// TIA Portal V18 program export: 0 tag tables, 0 data types, 87 data blocks, 42 code blocks (in call order from the OBs), 0 instance data blocks

DATA_BLOCK "DiagnosticDataBlock"
{ S7_Optimized_Access := 'FALSE' }
VERSION : 0.1
   STRUCT 
      DP : Struct
         DPReadStatus : Int;
         Status : Array[0..1023] of Bool;
      END_STRUCT;
      Profinet : Struct
         PNReadStatus : Int;
         Status : Array[0..1023] of Bool;
      END_STRUCT;
   END_STRUCT;


BEGIN

END_DATA_BLOCK

DATA_BLOCK "Sys"
{ S7_Optimized_Access := 'FALSE' }
VERSION : 0.1
   STRUCT 
      COM : Struct
         AlwaysOFF : Bool;
         AlwaysON : Bool;
         FlashTime100mS : Bool;
         FlashTime200mS : Bool;
         FlashTime500mS : Bool;
         FlashTime1S : Bool;
         FlashTime2S : Bool;
         SpareBit : Bool;
         PLCRestarted : Bool;
      END_STRUCT;
      SpareB1 : Array[0..7] of Byte;
      DateTime : Struct
         Set : Date_And_Time;
         Read : Date_And_Time;
         Trigger : Bool;
         ReturnValueRead : Int;
         ReturnValueSet : Int;
      END_STRUCT;
      SpareB2 : Array[0..17] of Byte;
      ScanTime : Struct
         CyclePrevious : Int;
         CycleMax : Int;
         CycleMin : Int;
      END_STRUCT;
      RETVALI : Int;
      RETVALW : Word;
      VersionManagement : Struct
         ProductLineName : String;
         ProjectNumber : String[20];
         "PLC IP Addr" : Array[0..3] of UInt;
         "HMI IP Addr" : Array[0..3] of UInt;
         PLCVersion : Array[0..1] of UInt;
         HMIVersion : Array[0..1] of UInt;
         "TIA Version" : String;
         StationID : Int;
         HMIPageID : Int;
      END_STRUCT;
   END_STRUCT;


BEGIN
   COM.AlwaysOFF := FALSE;
   COM.AlwaysON := TRUE;
   COM.FlashTime100mS := TRUE;
   COM.FlashTime200mS := TRUE;
   COM.FlashTime500mS := FALSE;
   COM.FlashTime1S := FALSE;
   COM.FlashTime2S := TRUE;
   COM.SpareBit := FALSE;
   COM.PLCRestarted := TRUE;
   SpareB1[0] := 16#00;
   SpareB1[1] := 16#00;
   SpareB1[2] := 16#00;
   SpareB1[3] := 16#00;
   SpareB1[4] := 16#00;
   SpareB1[5] := 16#00;
   SpareB1[6] := 16#00;
   SpareB1[7] := 16#00;
   DateTime.Set := DT#1990-01-01-00:00:00;
   DateTime.Read := DT#2025-03-12-08:03:05.785;
   DateTime.Trigger := FALSE;
   DateTime.ReturnValueRead := 0;
   DateTime.ReturnValueSet := 0;
   SpareB2[0] := 16#00;
   SpareB2[1] := 16#00;
   SpareB2[2] := 16#00;
   SpareB2[3] := 16#00;
   SpareB2[4] := 16#00;
   SpareB2[5] := 16#00;
   SpareB2[6] := 16#00;
   SpareB2[7] := 16#00;
   SpareB2[8] := 16#00;
   SpareB2[9] := 16#00;
   SpareB2[10] := 16#00;
   SpareB2[11] := 16#00;
   SpareB2[12] := 16#00;
   SpareB2[13] := 16#00;
   SpareB2[14] := 16#00;
   SpareB2[15] := 16#00;
   SpareB2[16] := 16#00;
   SpareB2[17] := 16#00;
   ScanTime.CyclePrevious := 14;
   ScanTime.CycleMax := 23;
   ScanTime.CycleMin := 9;
   RETVALI := 0;
   RETVALW := 16#0000;
   VersionManagement.ProductLineName := 'Assembly Line';
   VersionManagement.ProjectNumber := 'SZ23055';
   VersionManagement."PLC IP Addr"[0] := 192;
   VersionManagement."PLC IP Addr"[1] := 168;
   VersionManagement."PLC IP Addr"[2] := 10;
   VersionManagement."PLC IP Addr"[3] := 10;
   VersionManagement."HMI IP Addr"[0] := 192;
   VersionManagement."HMI IP Addr"[1] := 168;
   VersionManagement."HMI IP Addr"[2] := 45;
   VersionManagement."HMI IP Addr"[3] := 11;
   VersionManagement.PLCVersion[0] := 1;
   VersionManagement.PLCVersion[1] := 0;
   VersionManagement.HMIVersion[0] := 1;
   VersionManagement.HMIVersion[1] := 0;
   VersionManagement."TIA Version" := 'TIA V18';
   VersionManagement.StationID := 10;
   VersionManagement.HMIPageID := 0;

END_DATA_BLOCK

DATA_BLOCK "ST10_FB_Tower_4Lamp_DB"
{ S7_Optimized_Access := 'TRUE' }
VERSION : 0.1
NON_RETAIN
"FB_Tower_4Lamp"

BEGIN

END_DATA_BLOCK

DATA_BLOCK "ST10_SysOutput"
{ S7_Optimized_Access := 'TRUE' }
VERSION : 0.1
NON_RETAIN
   VAR 
      oTowerLight : Struct
         Red : Bool;
         Yellow : Bool;
         Green : Bool;
         Blue : Bool;
      END_STRUCT;
      HMIButtonLight : Struct
         ControlOn : Bool;
         ControlOff : Bool;
         MachineStart : Bool;
         MachineStop : Bool;
         ResetButton : Bool;
         "Manual/Auto" : Bool;
         SafetyGateUnlock : Bool;
      END_STRUCT;
      BoxLight : Struct
         oMachineStartLight : Bool;
         oMachineStopLight : Bool;
         oResetLight : Bool;
         oSafetyGateUnlockLight : Bool;
      END_STRUCT;
      SafetyDoorCoil : Array[1..20] of Bool;
      MaterialDoorCoil : Array[1..20] of Bool;
   END_VAR


BEGIN
   HMIButtonLight.ControlOn := false;
   HMIButtonLight.MachineStart := false;
   HMIButtonLight.MachineStop := false;
   HMIButtonLight.ResetButton := false;
   HMIButtonLight."Manual/Auto" := false;
   HMIButtonLight.SafetyGateUnlock := false;

END_DATA_BLOCK

DATA_BLOCK "AutoProcessData"
{ S7_Optimized_Access := 'FALSE' }
VERSION : 0.1
   STRUCT 
      A_ScanRotate { S7_SetPoint := 'False'} : "ProcessData";
      F_Robot1Grip1 : "ProcessData";
      F_Robot1Grip2 : "ProcessData";
      B_Press1 : "ProcessData";
      C_Glue : "ProcessData";
      F_Robot2Grip1 : "ProcessData";
      F_Robot2Grip2 : "ProcessData";
      C_GlueNGBuffer : "ProcessData";
      C_MagnScanNGBuffer : "ProcessData";
      B_Press2 : "ProcessData";
      F_Robot3Grip1 : "ProcessData";
      F_Robot3Grip2 : "ProcessData";
      H_ShafeLine : "ProcessData";
      J_ShafeLine : "ProcessData";
      K_ShafeLine : "ProcessData";
      L_ShafeLine : "ProcessData";
      ClearData : "ProcessData";
      A_Table_1 : Array[1..10] of "TableProcessData";
      A_Table_2 : Array[1..10] of "TableProcessData";
      FixtureCode_A1 { S7_SetPoint := 'True'} : Array[1..10] of String[128];
      FixtureCode_A2 { S7_SetPoint := 'True'} : Array[1..10] of String[128];
      GlobalData : Struct
         Table1CodeOKFlag : Bool;
         Table2CodeOKFlag : Bool;
         Fixture1CodeOKFlag : Bool;
         Fixture2CodeOKFlag : Bool;
         Robot2GripperCodeOKFlag : Bool;
         Robot1GripperCodeOKFlag : Bool;
         Robot3GripperCodeOKFlag : Bool;
         Spare_8 : Bool;
         Spare_9 : Bool;
         Spare_10 : Bool;
         Spare_11 : Bool;
         Spare_12 : Bool;
         Spare_13 : Bool;
         Spare_14 : Bool;
         Spare_15 : Bool;
         Spare_16 : Bool;
         DataIndex { S7_SetPoint := 'True'} : Int;
         Robot1GripCodeStatus1 : Int;
         Robot1GripCodeStatus2 : Int;
         Robot1GripCodeStatus3 : Int;
         Robot1GripCodeStatus4 : Int;
         Robot2GripCodeStatus1 : Int;
         Robot2GripCodeStatus2 : Int;
         Robot2GripCodeStatus3 : Int;
         Robot2GripCodeStatus4 : Int;
         Robot3GripCodeStatus1 : Int;
         Robot3GripCodeStatus2 : Int;
         Robot3GripCodeStatus3 : Int;
         Robot3GripCodeStatus4 : Int;
         FixtureCode_A1Status1 : Int;
         FixtureCode_A1Status2 : Int;
         FixtureCode_A1Status3 : Int;
         FixtureCode_A1Status4 : Int;
         FixtureCode_A1Status5 : Int;
         FixtureCode_A1Status6 : Int;
         FixtureCode_A1Status7 : Int;
         FixtureCode_A1Status8 : Int;
         FixtureCode_A1Status9 : Int;
         FixtureCode_A1Status10 : Int;
         FixtureCode_A2Status1 : Int;
         FixtureCode_A2Status2 : Int;
         FixtureCode_A2Status3 : Int;
         FixtureCode_A2Status4 : Int;
         FixtureCode_A2Status5 : Int;
         FixtureCode_A2Status6 : Int;
         FixtureCode_A2Status7 : Int;
         FixtureCode_A2Status8 : Int;
         FixtureCode_A2Status9 : Int;
         FixtureCode_A2Status10 : Int;
         Spare : Array[1..332] of Byte;
      END_STRUCT;
      DataBuffer { S7_SetPoint := 'False'} : Array[1..30] of "ProcessData";
      GripperCode_R1 { S7_SetPoint := 'True'} : Array[1..10] of String[128];
      GripperCode_R2 { S7_SetPoint := 'True'} : Array[1..10] of String[128];
      GripperCode_R3 { S7_SetPoint := 'True'} : Array[1..10] of String[128];
   END_STRUCT;


BEGIN
   A_Table_1[1].Code := 'SZ23055-OP010-E-Compressor-ring1 Loading tooling-1';
   A_Table_1[2].Code := 'SZ23055-OP010-E-Compressor-ring1 Loading tooling-2';
   A_Table_2[1].Code := 'SZ23055-OP010-E-Compressor-ring2 Loading tooling-1$R';
   GlobalData.DataIndex := 1;

END_DATA_BLOCK

DATA_BLOCK "PalletRelease"
{ S7_Optimized_Access := 'FALSE' }
VERSION : 0.1
NON_RETAIN
   STRUCT 
      Buffer : Struct
         AskPallet : Bool;
         UnloadFlag : Bool;
      END_STRUCT;
      LaserMarking : Struct
         AskPallet : Bool;
         UnloadFlag : Bool;
      END_STRUCT;
      Print : Struct
         AskPallet : Bool;
         UnloadFlag : Bool;
      END_STRUCT;
      Spare : Struct
         AskPallet : Bool;
         UnloadFlag : Bool;
      END_STRUCT;
      Spare2 : Struct
         AskPallet : Bool;
         UnloadFlag : Bool;
      END_STRUCT;
      "Time" {InstructionName := 'TOF_TIME'; LibVersion := '1.0'; S7_SetPoint := 'False'} : Array[0..1] of TOF_TIME;
      LaserMarkingBuffer { S7_SetPoint := 'False'} : "LaserMarkingBuffer";
   END_STRUCT;


BEGIN

END_DATA_BLOCK

DATA_BLOCK "ST10_GlobalError"
{ S7_Optimized_Access := 'FALSE' }
VERSION : 0.1
   STRUCT 
      COM : Struct
         MainPneumaticPressure1NOK : Bool;
         MainPneumaticPressure2NOK : Bool;
         MainPneumaticPressure3NOK : Bool;
         StationNotInHP : Bool;
         CabinetTemperatureNotOk : Bool;
         CoolingUnitNotOk : Bool;
         RotateTablePositionNOK : Bool;
         RotateTableNotInPosition : Bool;
         StationHardwareError : Bool;
         ChangeStyleError : Bool;
         Reserve3 : Bool;
         Reserve4 : Bool;
         Reserve5 : Bool;
         Reserve6 : Bool;
         Reserve7 : Bool;
         Reserve8 : Bool;
         Reserve : Array[1..4, 0..15] of Bool;
      END_STRUCT;
      Hardware : Struct
         PNSlaveStation01 : Array[1..10] of Struct
            Error : Bool;
            Reserve1 : Bool;
            Reserve2 : Bool;
         END_STRUCT;
         COMM : Array[1..5] of Struct
            CommunicationError : Bool;
            NoReceive : Bool;
            ReceiveWrong : Bool;
            Reserve1 : Bool;
            Reserve2 : Bool;
         END_STRUCT;
         PNSlaveStation02 : Array[1..10] of Struct
            Error : Bool;
            Reserve1 : Bool;
            Reserve2 : Bool;
            Reserve3 : Bool;
         END_STRUCT;
         PNSlaveStation03 : Array[1..10] of Struct
            Error : Bool;
            Reserve1 : Bool;
            Reserve2 : Bool;
            Reserve3 : Bool;
         END_STRUCT;
         ValveIsland : Array[1..5] of Struct
            SystemError : Bool;
            OffLine : Bool;
            Reserve1 : Bool;
            Reserve2 : Bool;
         END_STRUCT;
      END_STRUCT;
      Safety : Struct
         "Robot 1 Estop" : Bool;
         "Robot 2 Estop" : Bool;
         HMIEstopPBActivated : Bool;
         TableEstopPB1Activated : Bool;
         TableEstopPB2Activated : Bool;
         TableEstopPB3Activated : Bool;
         TableEstopPB4Activated : Bool;
         TableEstopPB5Activated : Bool;
         TableEstopPB6Activated : Bool;
         EStopSafety : Bool;
         TableEstopPB7Activated : Bool;
         TableEstopPB8Activated : Bool;
         TableEstopPB9Activated : Bool;
         StoveEstopActivated : Bool;
         "Robot 3 Estop" : Bool;
         Reserve9 : Bool;
         Reserve : Array[1..4, 0..15] of Bool;
      END_STRUCT;
      SafetyDoor : Struct
         "Type" : Array[1..5] of Struct
            NotOk : Bool;
            OpenInRunning : Bool;
            Reserve1 : Bool;
            Reserve2 : Bool;
         END_STRUCT;
         No : Array[1..9] of Struct
            NotLock : Bool;
            Notlocked : Bool;
            NotClose : Bool;
            Reserve1 : Bool;
            Reserve2 : Bool;
         END_STRUCT;
         MaterialDoor : Struct
            NotLock_1 : Bool;
            NotClose_1 : Bool;
            NotLock_2 : Bool;
            NotClose_2 : Bool;
            NotLock_3 : Bool;
            NotClose_3 : Bool;
            NotLock_4 : Bool;
            NotClose_4 : Bool;
            NotLock_5 : Bool;
            NotClose_5 : Bool;
            NotLock_6 : Bool;
            NotClose_6 : Bool;
            NotLock_7 : Bool;
            NotClose_7 : Bool;
            NotLock_8 : Bool;
            NotClose_8 : Bool;
         END_STRUCT;
      END_STRUCT;
      LightCurtain : Array[1..5] of Struct
         ActivatedInRunning : Bool;
         ActivatedInRotTableRun : Bool;
         Error : Bool;
         Reserve1 : Bool;
         Reserve2 : Bool;
      END_STRUCT;
      Product : Array[1..5] of Struct
         TypeSelectionError : Bool;
         TypeWrong : Bool;
         NotforStation : Bool;
         TypeAutoChangeError : Bool;
         Reserve2 : Bool;
      END_STRUCT;
      Fixture : Array[1..10] of Struct
         PositionError : Bool;
         TypeError : Bool;
         Reserve1 : Bool;
         Reserve2 : Bool;
      END_STRUCT;
      Breaker : Struct
         Trip : Array[1..16] of Bool;
      END_STRUCT;
   END_STRUCT;


BEGIN

END_DATA_BLOCK

DATA_BLOCK "ST10_TipDB"
{ S7_Optimized_Access := 'FALSE' }
VERSION : 0.1
   STRUCT 
      Global : Struct
         "1" : Struct
            ControlOn : Bool;
            closesafetyDoor : Bool;
            LockSafetyDoor : Bool;
            SelectAutoMode : Bool;
            SelectManualMode : Bool;
            AutoModeRunning : Bool;
            SafetyDoorLocked : Bool;
            SaferyDoorNotLocked : Bool;
            GoWP : Bool;
            Reset : Bool;
         END_STRUCT;
         "2" : Array[0..15] of Bool;
         "3" : Array[0..15] of Bool;
         "4" : Array[0..15] of Bool;
         "5" : Struct
            FuncrionDeactive1 : Bool;
            FuncrionDeactive2 : Bool;
            FuncrionDeactive3 : Bool;
            FuncrionDeactive4 : Bool;
            FuncrionDeactive5 : Bool;
            FuncrionDeactive6 : Bool;
            FuncrionDeactive7 : Bool;
            FuncrionDeactive8 : Bool;
         END_STRUCT;
         "6" : Array[0..15] of Bool;
         "7" : Struct
            ScanMainPartDMC1 : Bool;
            ScanPartDMC2 : Bool;
            ScanPartDMC3 : Bool;
            ScanPartDMC4 : Bool;
            ScanPartDMC5 : Bool;
            ScanPartDMC6 : Bool;
            ScanPartDMC7 : Bool;
            ScanPartDMC8 : Bool;
         END_STRUCT;
         "8" : Array[0..15] of Bool;
         "9" : Array[0..15] of Bool;
         "10" : Array[0..15] of Bool;
      END_STRUCT;
      OP1 : Struct
         "Take off product" : Bool;
         "Put product" : Bool;
         "Please scan the code" : Bool;
         "Please apply Oil" : Bool;
         "Please take the O-ring" : Bool;
         "Please put in the powertrain" : Bool;
         Static_2 : Bool;
         "Please pre-screw" : Bool;
         Static_1 : Bool;
         Static_3 : Bool;
         "Please press the button_1" : Bool;
         Reset : Bool;
      END_STRUCT;
      OP2 : Struct
         Static_4 : Bool;
         Static_2 : Bool;
         Static_3 : Bool;
         "Please press the button" : Bool;
         "Please press the trigger" : Bool;
         "Please take the paint pen" : Bool;
         "Please put back the paint pen" : Bool;
         Static_1 : Bool;
         "Please remove the product" : Bool;
         "Please press the screw gun trigger" : Bool;
      END_STRUCT;
   END_STRUCT;


BEGIN

END_DATA_BLOCK

DATA_BLOCK "Parameter"
{ S7_Optimized_Access := 'TRUE' }
VERSION : 0.1
NON_RETAIN
   VAR RETAIN
      AxisRun : Struct
         Axis { S7_SetPoint := 'False'} : Array[1..15] of "ServoType_UDT";
      END_STRUCT;
      AxisNuw : Struct
         Axis { S7_SetPoint := 'False'} : Array[1..15] of "ServoType_UDT";
      END_STRUCT;
      AxisDisplay : Struct
         Axis { S7_SetPoint := 'False'} : Array[1..15] of "ServoType_UDT";
      END_STRUCT;
      AxisSave : Struct
         Axis { S7_SetPoint := 'False'} : Array[1..15] of "ServoType_UDT";
      END_STRUCT;
      AxisStore : Array[1..15] of Struct
         Axis { S7_SetPoint := 'False'} : Array[1..15] of "ServoType_UDT";
      END_STRUCT;
   END_VAR


BEGIN
   AxisRun.Axis[1].Pos1.Position := 3.419;
   AxisRun.Axis[1].Pos1.Speed := 10000;
   AxisRun.Axis[1].Pos1.Reached := FALSE;
   AxisRun.Axis[1].Pos2.Position := 48.386;
   AxisRun.Axis[1].Pos2.Speed := 10000;
   AxisRun.Axis[1].Pos2.Reached := FALSE;
   AxisRun.Axis[1].Pos3.Position := 93.294;
   AxisRun.Axis[1].Pos3.Speed := 10000;
   AxisRun.Axis[1].Pos3.Reached := FALSE;
   AxisRun.Axis[1].Pos4.Position := 138.335;
   AxisRun.Axis[1].Pos4.Speed := 10000;
   AxisRun.Axis[1].Pos4.Reached := FALSE;
   AxisRun.Axis[1].Pos5.Position := 183.464;
   AxisRun.Axis[1].Pos5.Speed := 10000;
   AxisRun.Axis[1].Pos5.Reached := FALSE;
   AxisRun.Axis[1].Pos6.Position := 228.443;
   AxisRun.Axis[1].Pos6.Speed := 10000;
   AxisRun.Axis[1].Pos6.Reached := FALSE;
   AxisRun.Axis[1].Pos7.Position := 273.535;
   AxisRun.Axis[1].Pos7.Speed := 10000;
   AxisRun.Axis[1].Pos7.Reached := FALSE;
   AxisRun.Axis[1].Pos8.Position := 318.25;
   AxisRun.Axis[1].Pos8.Speed := 10000;
   AxisRun.Axis[1].Pos8.Reached := FALSE;
   AxisRun.Axis[1].Pos9.Position := 0.0;
   AxisRun.Axis[1].Pos9.Speed := 0;
   AxisRun.Axis[1].Pos9.Reached := FALSE;
   AxisRun.Axis[1].Pos10.Position := 0.0;
   AxisRun.Axis[1].Pos10.Speed := 0;
   AxisRun.Axis[1].Pos10.Reached := FALSE;
   AxisRun.Axis[1].Pos11.Position := 0.0;
   AxisRun.Axis[1].Pos11.Speed := 0;
   AxisRun.Axis[1].Pos11.Reached := FALSE;
   AxisRun.Axis[1].Pos12.Position := 0.0;
   AxisRun.Axis[1].Pos12.Speed := 0;
   AxisRun.Axis[1].Pos12.Reached := FALSE;
   AxisRun.Axis[1].Pos13.Position := 0.0;
   AxisRun.Axis[1].Pos13.Speed := 0;
   AxisRun.Axis[1].Pos13.Reached := FALSE;
   AxisRun.Axis[1].Pos14.Position := 0.0;
   AxisRun.Axis[1].Pos14.Speed := 0;
   AxisRun.Axis[1].Pos14.Reached := FALSE;
   AxisRun.Axis[1].Pos15.Position := 0.0;
   AxisRun.Axis[1].Pos15.Speed := 0;
   AxisRun.Axis[1].Pos15.Reached := FALSE;
   AxisRun.Axis[1].Pos16.Position := 0.0;
   AxisRun.Axis[1].Pos16.Speed := 0;
   AxisRun.Axis[1].Pos16.Reached := FALSE;
   AxisRun.Axis[1].Pos17.Position := 0.0;
   AxisRun.Axis[1].Pos17.Speed := 0;
   AxisRun.Axis[1].Pos17.Reached := FALSE;
   AxisRun.Axis[1].Pos18.Position := 0.0;
   AxisRun.Axis[1].Pos18.Speed := 0;
   AxisRun.Axis[1].Pos18.Reached := FALSE;
   AxisRun.Axis[1].Pos19.Position := 0.0;
   AxisRun.Axis[1].Pos19.Speed := 0;
   AxisRun.Axis[1].Pos19.Reached := FALSE;
   AxisRun.Axis[1].Pos20.Position := 0.0;
   AxisRun.Axis[1].Pos20.Speed := 0;
   AxisRun.Axis[1].Pos20.Reached := FALSE;
   AxisRun.Axis[1].Pos21.Position := 0.0;
   AxisRun.Axis[1].Pos21.Speed := 0;
   AxisRun.Axis[1].Pos21.Reached := FALSE;
   AxisRun.Axis[1].Pos22.Position := 0.0;
   AxisRun.Axis[1].Pos22.Speed := 0;
   AxisRun.Axis[1].Pos22.Reached := FALSE;
   AxisRun.Axis[1].Pos23.Position := 0.0;
   AxisRun.Axis[1].Pos23.Speed := 0;
   AxisRun.Axis[1].Pos23.Reached := FALSE;
   AxisRun.Axis[1].Pos24.Position := 0.0;
   AxisRun.Axis[1].Pos24.Speed := 0;
   AxisRun.Axis[1].Pos24.Reached := FALSE;
   AxisRun.Axis[1].Pos25.Position := 0.0;
   AxisRun.Axis[1].Pos25.Speed := 0;
   AxisRun.Axis[1].Pos25.Reached := FALSE;
   AxisRun.Axis[1].Pos26.Position := 0.0;
   AxisRun.Axis[1].Pos26.Speed := 0;
   AxisRun.Axis[1].Pos26.Reached := FALSE;
   AxisRun.Axis[1].Pos27.Position := 0.0;
   AxisRun.Axis[1].Pos27.Speed := 0;
   AxisRun.Axis[1].Pos27.Reached := FALSE;
   AxisRun.Axis[1].Pos28.Position := 0.0;
   AxisRun.Axis[1].Pos28.Speed := 0;
   AxisRun.Axis[1].Pos28.Reached := FALSE;
   AxisRun.Axis[1].Pos29.Position := 0.0;
   AxisRun.Axis[1].Pos29.Speed := 0;
   AxisRun.Axis[1].Pos29.Reached := FALSE;
   AxisRun.Axis[1].Pos30.Position := 0.0;
   AxisRun.Axis[1].Pos30.Speed := 0;
   AxisRun.Axis[1].Pos30.Reached := FALSE;
   AxisRun.Axis[2].Pos1.Position := 0.0;
   AxisRun.Axis[2].Pos1.Speed := 10000;
   AxisRun.Axis[2].Pos1.Reached := FALSE;
   AxisRun.Axis[2].Pos2.Position := 450.0;
   AxisRun.Axis[2].Pos2.Speed := 10000;
   AxisRun.Axis[2].Pos2.Reached := FALSE;
   AxisRun.Axis[2].Pos3.Position := 900.0;
   AxisRun.Axis[2].Pos3.Speed := 10000;
   AxisRun.Axis[2].Pos3.Reached := FALSE;
   AxisRun.Axis[2].Pos4.Position := 135.0;
   AxisRun.Axis[2].Pos4.Speed := 10000;
   AxisRun.Axis[2].Pos4.Reached := FALSE;
   AxisRun.Axis[2].Pos5.Position := 180.0;
   AxisRun.Axis[2].Pos5.Speed := 10000;
   AxisRun.Axis[2].Pos5.Reached := FALSE;
   AxisRun.Axis[2].Pos6.Position := 225.0;
   AxisRun.Axis[2].Pos6.Speed := 10000;
   AxisRun.Axis[2].Pos6.Reached := FALSE;
   AxisRun.Axis[2].Pos7.Position := 270.0;
   AxisRun.Axis[2].Pos7.Speed := 10000;
   AxisRun.Axis[2].Pos7.Reached := FALSE;
   AxisRun.Axis[2].Pos8.Position := 315.0;
   AxisRun.Axis[2].Pos8.Speed := 10000;
   AxisRun.Axis[2].Pos8.Reached := FALSE;
   AxisRun.Axis[2].Pos9.Position := 0.0;
   AxisRun.Axis[2].Pos9.Speed := 0;
   AxisRun.Axis[2].Pos9.Reached := FALSE;
   AxisRun.Axis[2].Pos10.Position := 0.0;
   AxisRun.Axis[2].Pos10.Speed := 0;
   AxisRun.Axis[2].Pos10.Reached := FALSE;
   AxisRun.Axis[2].Pos11.Position := 0.0;
   AxisRun.Axis[2].Pos11.Speed := 0;
   AxisRun.Axis[2].Pos11.Reached := FALSE;
   AxisRun.Axis[2].Pos12.Position := 0.0;
   AxisRun.Axis[2].Pos12.Speed := 0;
   AxisRun.Axis[2].Pos12.Reached := FALSE;
   AxisRun.Axis[2].Pos13.Position := 0.0;
   AxisRun.Axis[2].Pos13.Speed := 0;
   AxisRun.Axis[2].Pos13.Reached := FALSE;
   AxisRun.Axis[2].Pos14.Position := 0.0;
   AxisRun.Axis[2].Pos14.Speed := 0;
   AxisRun.Axis[2].Pos14.Reached := FALSE;
   AxisRun.Axis[2].Pos15.Position := 0.0;
   AxisRun.Axis[2].Pos15.Speed := 0;
   AxisRun.Axis[2].Pos15.Reached := FALSE;
   AxisRun.Axis[2].Pos16.Position := 0.0;
   AxisRun.Axis[2].Pos16.Speed := 0;
   AxisRun.Axis[2].Pos16.Reached := FALSE;
   AxisRun.Axis[2].Pos17.Position := 0.0;
   AxisRun.Axis[2].Pos17.Speed := 0;
   AxisRun.Axis[2].Pos17.Reached := FALSE;
   AxisRun.Axis[2].Pos18.Position := 0.0;
   AxisRun.Axis[2].Pos18.Speed := 0;
   AxisRun.Axis[2].Pos18.Reached := FALSE;
   AxisRun.Axis[2].Pos19.Position := 0.0;
   AxisRun.Axis[2].Pos19.Speed := 0;
   AxisRun.Axis[2].Pos19.Reached := FALSE;
   AxisRun.Axis[2].Pos20.Position := 0.0;
   AxisRun.Axis[2].Pos20.Speed := 0;
   AxisRun.Axis[2].Pos20.Reached := FALSE;
   AxisRun.Axis[2].Pos21.Position := 0.0;
   AxisRun.Axis[2].Pos21.Speed := 0;
   AxisRun.Axis[2].Pos21.Reached := FALSE;
   AxisRun.Axis[2].Pos22.Position := 0.0;
   AxisRun.Axis[2].Pos22.Speed := 0;
   AxisRun.Axis[2].Pos22.Reached := FALSE;
   AxisRun.Axis[2].Pos23.Position := 0.0;
   AxisRun.Axis[2].Pos23.Speed := 0;
   AxisRun.Axis[2].Pos23.Reached := FALSE;
   AxisRun.Axis[2].Pos24.Position := 0.0;
   AxisRun.Axis[2].Pos24.Speed := 0;
   AxisRun.Axis[2].Pos24.Reached := FALSE;
   AxisRun.Axis[2].Pos25.Position := 0.0;
   AxisRun.Axis[2].Pos25.Speed := 0;
   AxisRun.Axis[2].Pos25.Reached := FALSE;
   AxisRun.Axis[2].Pos26.Position := 0.0;
   AxisRun.Axis[2].Pos26.Speed := 0;
   AxisRun.Axis[2].Pos26.Reached := FALSE;
   AxisRun.Axis[2].Pos27.Position := 0.0;
   AxisRun.Axis[2].Pos27.Speed := 0;
   AxisRun.Axis[2].Pos27.Reached := FALSE;
   AxisRun.Axis[2].Pos28.Position := 0.0;
   AxisRun.Axis[2].Pos28.Speed := 0;
   AxisRun.Axis[2].Pos28.Reached := FALSE;
   AxisRun.Axis[2].Pos29.Position := 0.0;
   AxisRun.Axis[2].Pos29.Speed := 0;
   AxisRun.Axis[2].Pos29.Reached := FALSE;
   AxisRun.Axis[2].Pos30.Position := 0.0;
   AxisRun.Axis[2].Pos30.Speed := 0;
   AxisRun.Axis[2].Pos30.Reached := FALSE;
   AxisRun.Axis[3].Pos1.Position := 0.0;
   AxisRun.Axis[3].Pos1.Speed := 20000;
   AxisRun.Axis[3].Pos1.Reached := FALSE;
   AxisRun.Axis[3].Pos2.Position := 490.0;
   AxisRun.Axis[3].Pos2.Speed := 10000;
   AxisRun.Axis[3].Pos2.Reached := FALSE;
   AxisRun.Axis[3].Pos3.Position := 490.0;
   AxisRun.Axis[3].Pos3.Speed := 10000;
   AxisRun.Axis[3].Pos3.Reached := FALSE;
   AxisRun.Axis[3].Pos4.Position := 490.0;
   AxisRun.Axis[3].Pos4.Speed := 10000;
   AxisRun.Axis[3].Pos4.Reached := FALSE;
   AxisRun.Axis[3].Pos5.Position := 0.0;
   AxisRun.Axis[3].Pos5.Speed := 0;
   AxisRun.Axis[3].Pos5.Reached := FALSE;
   AxisRun.Axis[3].Pos6.Position := 490.0;
   AxisRun.Axis[3].Pos6.Speed := 10000;
   AxisRun.Axis[3].Pos6.Reached := FALSE;
   AxisRun.Axis[3].Pos7.Position := 90.0;
   AxisRun.Axis[3].Pos7.Speed := 10000;
   AxisRun.Axis[3].Pos7.Reached := FALSE;
   AxisRun.Axis[3].Pos8.Position := 180.0;
   AxisRun.Axis[3].Pos8.Speed := 10000;
   AxisRun.Axis[3].Pos8.Reached := FALSE;
   AxisRun.Axis[3].Pos9.Position := 270.0;
   AxisRun.Axis[3].Pos9.Speed := 10000;
   AxisRun.Axis[3].Pos9.Reached := FALSE;
   AxisRun.Axis[3].Pos10.Position := 0.0;
   AxisRun.Axis[3].Pos10.Speed := 0;
   AxisRun.Axis[3].Pos10.Reached := FALSE;
   AxisRun.Axis[3].Pos11.Position := 0.0;
   AxisRun.Axis[3].Pos11.Speed := 0;
   AxisRun.Axis[3].Pos11.Reached := FALSE;
   AxisRun.Axis[3].Pos12.Position := 0.0;
   AxisRun.Axis[3].Pos12.Speed := 0;
   AxisRun.Axis[3].Pos12.Reached := FALSE;
   AxisRun.Axis[3].Pos13.Position := 0.0;
   AxisRun.Axis[3].Pos13.Speed := 0;
   AxisRun.Axis[3].Pos13.Reached := FALSE;
   AxisRun.Axis[3].Pos14.Position := 0.0;
   AxisRun.Axis[3].Pos14.Speed := 0;
   AxisRun.Axis[3].Pos14.Reached := FALSE;
   AxisRun.Axis[3].Pos15.Position := 0.0;
   AxisRun.Axis[3].Pos15.Speed := 0;
   AxisRun.Axis[3].Pos15.Reached := FALSE;
   AxisRun.Axis[3].Pos16.Position := 0.0;
   AxisRun.Axis[3].Pos16.Speed := 0;
   AxisRun.Axis[3].Pos16.Reached := FALSE;
   AxisRun.Axis[3].Pos17.Position := 0.0;
   AxisRun.Axis[3].Pos17.Speed := 0;
   AxisRun.Axis[3].Pos17.Reached := FALSE;
   AxisRun.Axis[3].Pos18.Position := 0.0;
   AxisRun.Axis[3].Pos18.Speed := 0;
   AxisRun.Axis[3].Pos18.Reached := FALSE;
   AxisRun.Axis[3].Pos19.Position := 0.0;
   AxisRun.Axis[3].Pos19.Speed := 0;
   AxisRun.Axis[3].Pos19.Reached := FALSE;
   AxisRun.Axis[3].Pos20.Position := 0.0;
   AxisRun.Axis[3].Pos20.Speed := 0;
   AxisRun.Axis[3].Pos20.Reached := FALSE;
   AxisRun.Axis[3].Pos21.Position := 0.0;
   AxisRun.Axis[3].Pos21.Speed := 0;
   AxisRun.Axis[3].Pos21.Reached := FALSE;
   AxisRun.Axis[3].Pos22.Position := 0.0;
   AxisRun.Axis[3].Pos22.Speed := 0;
   AxisRun.Axis[3].Pos22.Reached := FALSE;
   AxisRun.Axis[3].Pos23.Position := 0.0;
   AxisRun.Axis[3].Pos23.Speed := 0;
   AxisRun.Axis[3].Pos23.Reached := FALSE;
   AxisRun.Axis[3].Pos24.Position := 0.0;
   AxisRun.Axis[3].Pos24.Speed := 0;
   AxisRun.Axis[3].Pos24.Reached := FALSE;
   AxisRun.Axis[3].Pos25.Position := 0.0;
   AxisRun.Axis[3].Pos25.Speed := 0;
   AxisRun.Axis[3].Pos25.Reached := FALSE;
   AxisRun.Axis[3].Pos26.Position := 0.0;
   AxisRun.Axis[3].Pos26.Speed := 0;
   AxisRun.Axis[3].Pos26.Reached := FALSE;
   AxisRun.Axis[3].Pos27.Position := 0.0;
   AxisRun.Axis[3].Pos27.Speed := 0;
   AxisRun.Axis[3].Pos27.Reached := FALSE;
   AxisRun.Axis[3].Pos28.Position := 0.0;
   AxisRun.Axis[3].Pos28.Speed := 0;
   AxisRun.Axis[3].Pos28.Reached := FALSE;
   AxisRun.Axis[3].Pos29.Position := 0.0;
   AxisRun.Axis[3].Pos29.Speed := 0;
   AxisRun.Axis[3].Pos29.Reached := FALSE;
   AxisRun.Axis[3].Pos30.Position := 0.0;
   AxisRun.Axis[3].Pos30.Speed := 0;
   AxisRun.Axis[3].Pos30.Reached := FALSE;
   AxisRun.Axis[4].Pos1.Position := 3.585;
   AxisRun.Axis[4].Pos1.Speed := 10000;
   AxisRun.Axis[4].Pos1.Reached := FALSE;
   AxisRun.Axis[4].Pos2.Position := 48.61;
   AxisRun.Axis[4].Pos2.Speed := 10000;
   AxisRun.Axis[4].Pos2.Reached := FALSE;
   AxisRun.Axis[4].Pos3.Position := 93.637;
   AxisRun.Axis[4].Pos3.Speed := 10000;
   AxisRun.Axis[4].Pos3.Reached := FALSE;
   AxisRun.Axis[4].Pos4.Position := 138.606;
   AxisRun.Axis[4].Pos4.Speed := 10000;
   AxisRun.Axis[4].Pos4.Reached := FALSE;
   AxisRun.Axis[4].Pos5.Position := 183.388;
   AxisRun.Axis[4].Pos5.Speed := 10000;
   AxisRun.Axis[4].Pos5.Reached := FALSE;
   AxisRun.Axis[4].Pos6.Position := 228.458;
   AxisRun.Axis[4].Pos6.Speed := 10000;
   AxisRun.Axis[4].Pos6.Reached := FALSE;
   AxisRun.Axis[4].Pos7.Position := 273.513;
   AxisRun.Axis[4].Pos7.Speed := 10000;
   AxisRun.Axis[4].Pos7.Reached := FALSE;
   AxisRun.Axis[4].Pos8.Position := 318.501;
   AxisRun.Axis[4].Pos8.Speed := 10000;
   AxisRun.Axis[4].Pos8.Reached := FALSE;
   AxisRun.Axis[4].Pos9.Position := 0.0;
   AxisRun.Axis[4].Pos9.Speed := 0;
   AxisRun.Axis[4].Pos9.Reached := FALSE;
   AxisRun.Axis[4].Pos10.Position := 0.0;
   AxisRun.Axis[4].Pos10.Speed := 0;
   AxisRun.Axis[4].Pos10.Reached := FALSE;
   AxisRun.Axis[4].Pos11.Position := 0.0;
   AxisRun.Axis[4].Pos11.Speed := 0;
   AxisRun.Axis[4].Pos11.Reached := FALSE;
   AxisRun.Axis[4].Pos12.Position := 0.0;
   AxisRun.Axis[4].Pos12.Speed := 0;
   AxisRun.Axis[4].Pos12.Reached := FALSE;
   AxisRun.Axis[4].Pos13.Position := 0.0;
   AxisRun.Axis[4].Pos13.Speed := 0;
   AxisRun.Axis[4].Pos13.Reached := FALSE;
   AxisRun.Axis[4].Pos14.Position := 0.0;
   AxisRun.Axis[4].Pos14.Speed := 0;
   AxisRun.Axis[4].Pos14.Reached := FALSE;
   AxisRun.Axis[4].Pos15.Position := 0.0;
   AxisRun.Axis[4].Pos15.Speed := 0;
   AxisRun.Axis[4].Pos15.Reached := FALSE;
   AxisRun.Axis[4].Pos16.Position := 0.0;
   AxisRun.Axis[4].Pos16.Speed := 0;
   AxisRun.Axis[4].Pos16.Reached := FALSE;
   AxisRun.Axis[4].Pos17.Position := 0.0;
   AxisRun.Axis[4].Pos17.Speed := 0;
   AxisRun.Axis[4].Pos17.Reached := FALSE;
   AxisRun.Axis[4].Pos18.Position := 0.0;
   AxisRun.Axis[4].Pos18.Speed := 0;
   AxisRun.Axis[4].Pos18.Reached := FALSE;
   AxisRun.Axis[4].Pos19.Position := 0.0;
   AxisRun.Axis[4].Pos19.Speed := 0;
   AxisRun.Axis[4].Pos19.Reached := FALSE;
   AxisRun.Axis[4].Pos20.Position := 0.0;
   AxisRun.Axis[4].Pos20.Speed := 0;
   AxisRun.Axis[4].Pos20.Reached := FALSE;
   AxisRun.Axis[4].Pos21.Position := 0.0;
   AxisRun.Axis[4].Pos21.Speed := 0;
   AxisRun.Axis[4].Pos21.Reached := FALSE;
   AxisRun.Axis[4].Pos22.Position := 0.0;
   AxisRun.Axis[4].Pos22.Speed := 0;
   AxisRun.Axis[4].Pos22.Reached := FALSE;
   AxisRun.Axis[4].Pos23.Position := 0.0;
   AxisRun.Axis[4].Pos23.Speed := 0;
   AxisRun.Axis[4].Pos23.Reached := FALSE;
   AxisRun.Axis[4].Pos24.Position := 0.0;
   AxisRun.Axis[4].Pos24.Speed := 0;
   AxisRun.Axis[4].Pos24.Reached := FALSE;
   AxisRun.Axis[4].Pos25.Position := 0.0;
   AxisRun.Axis[4].Pos25.Speed := 0;
   AxisRun.Axis[4].Pos25.Reached := FALSE;
   AxisRun.Axis[4].Pos26.Position := 0.0;
   AxisRun.Axis[4].Pos26.Speed := 0;
   AxisRun.Axis[4].Pos26.Reached := FALSE;
   AxisRun.Axis[4].Pos27.Position := 0.0;
   AxisRun.Axis[4].Pos27.Speed := 0;
   AxisRun.Axis[4].Pos27.Reached := FALSE;
   AxisRun.Axis[4].Pos28.Position := 0.0;
   AxisRun.Axis[4].Pos28.Speed := 0;
   AxisRun.Axis[4].Pos28.Reached := FALSE;
   AxisRun.Axis[4].Pos29.Position := 0.0;
   AxisRun.Axis[4].Pos29.Speed := 0;
   AxisRun.Axis[4].Pos29.Reached := FALSE;
   AxisRun.Axis[4].Pos30.Position := 0.0;
   AxisRun.Axis[4].Pos30.Speed := 0;
   AxisRun.Axis[4].Pos30.Reached := FALSE;
   AxisRun.Axis[5].Pos1.Position := 143.76;
   AxisRun.Axis[5].Pos1.Speed := 200;
   AxisRun.Axis[5].Pos1.Reached := FALSE;
   AxisRun.Axis[5].Pos2.Position := 143.76;
   AxisRun.Axis[5].Pos2.Speed := 200;
   AxisRun.Axis[5].Pos2.Reached := FALSE;
   AxisRun.Axis[5].Pos3.Position := 137.76;
   AxisRun.Axis[5].Pos3.Speed := 200;
   AxisRun.Axis[5].Pos3.Reached := FALSE;
   AxisRun.Axis[5].Pos4.Position := 130.36;
   AxisRun.Axis[5].Pos4.Speed := 200;
   AxisRun.Axis[5].Pos4.Reached := FALSE;
   AxisRun.Axis[5].Pos5.Position := 124.16;
   AxisRun.Axis[5].Pos5.Speed := 200;
   AxisRun.Axis[5].Pos5.Reached := FALSE;
   AxisRun.Axis[5].Pos6.Position := 125.65;
   AxisRun.Axis[5].Pos6.Speed := 200;
   AxisRun.Axis[5].Pos6.Reached := FALSE;
   AxisRun.Axis[5].Pos7.Position := 48.11;
   AxisRun.Axis[5].Pos7.Speed := 200;
   AxisRun.Axis[5].Pos7.Reached := FALSE;
   AxisRun.Axis[5].Pos8.Position := 0.0;
   AxisRun.Axis[5].Pos8.Speed := 200;
   AxisRun.Axis[5].Pos8.Reached := FALSE;
   AxisRun.Axis[5].Pos9.Position := 48.11;
   AxisRun.Axis[5].Pos9.Speed := 200;
   AxisRun.Axis[5].Pos9.Reached := FALSE;
   AxisRun.Axis[5].Pos10.Position := 0.0;
   AxisRun.Axis[5].Pos10.Speed := 0;
   AxisRun.Axis[5].Pos10.Reached := FALSE;
   AxisRun.Axis[5].Pos11.Position := 0.0;
   AxisRun.Axis[5].Pos11.Speed := 0;
   AxisRun.Axis[5].Pos11.Reached := FALSE;
   AxisRun.Axis[5].Pos12.Position := 0.0;
   AxisRun.Axis[5].Pos12.Speed := 0;
   AxisRun.Axis[5].Pos12.Reached := FALSE;
   AxisRun.Axis[5].Pos13.Position := 0.0;
   AxisRun.Axis[5].Pos13.Speed := 0;
   AxisRun.Axis[5].Pos13.Reached := FALSE;
   AxisRun.Axis[5].Pos14.Position := 0.0;
   AxisRun.Axis[5].Pos14.Speed := 0;
   AxisRun.Axis[5].Pos14.Reached := FALSE;
   AxisRun.Axis[5].Pos15.Position := 0.0;
   AxisRun.Axis[5].Pos15.Speed := 0;
   AxisRun.Axis[5].Pos15.Reached := FALSE;
   AxisRun.Axis[5].Pos16.Position := 0.0;
   AxisRun.Axis[5].Pos16.Speed := 0;
   AxisRun.Axis[5].Pos16.Reached := FALSE;
   AxisRun.Axis[5].Pos17.Position := 0.0;
   AxisRun.Axis[5].Pos17.Speed := 0;
   AxisRun.Axis[5].Pos17.Reached := FALSE;
   AxisRun.Axis[5].Pos18.Position := 0.0;
   AxisRun.Axis[5].Pos18.Speed := 0;
   AxisRun.Axis[5].Pos18.Reached := FALSE;
   AxisRun.Axis[5].Pos19.Position := 0.0;
   AxisRun.Axis[5].Pos19.Speed := 0;
   AxisRun.Axis[5].Pos19.Reached := FALSE;
   AxisRun.Axis[5].Pos20.Position := 0.0;
   AxisRun.Axis[5].Pos20.Speed := 0;
   AxisRun.Axis[5].Pos20.Reached := FALSE;
   AxisRun.Axis[5].Pos21.Position := 0.0;
   AxisRun.Axis[5].Pos21.Speed := 0;
   AxisRun.Axis[5].Pos21.Reached := FALSE;
   AxisRun.Axis[5].Pos22.Position := 0.0;
   AxisRun.Axis[5].Pos22.Speed := 0;
   AxisRun.Axis[5].Pos22.Reached := FALSE;
   AxisRun.Axis[5].Pos23.Position := 0.0;
   AxisRun.Axis[5].Pos23.Speed := 0;
   AxisRun.Axis[5].Pos23.Reached := FALSE;
   AxisRun.Axis[5].Pos24.Position := 0.0;
   AxisRun.Axis[5].Pos24.Speed := 0;
   AxisRun.Axis[5].Pos24.Reached := FALSE;
   AxisRun.Axis[5].Pos25.Position := 0.0;
   AxisRun.Axis[5].Pos25.Speed := 0;
   AxisRun.Axis[5].Pos25.Reached := FALSE;
   AxisRun.Axis[5].Pos26.Position := 0.0;
   AxisRun.Axis[5].Pos26.Speed := 0;
   AxisRun.Axis[5].Pos26.Reached := FALSE;
   AxisRun.Axis[5].Pos27.Position := 0.0;
   AxisRun.Axis[5].Pos27.Speed := 0;
   AxisRun.Axis[5].Pos27.Reached := FALSE;
   AxisRun.Axis[5].Pos28.Position := 0.0;
   AxisRun.Axis[5].Pos28.Speed := 0;
   AxisRun.Axis[5].Pos28.Reached := FALSE;
   AxisRun.Axis[5].Pos29.Position := 0.0;
   AxisRun.Axis[5].Pos29.Speed := 0;
   AxisRun.Axis[5].Pos29.Reached := FALSE;
   AxisRun.Axis[5].Pos30.Position := 0.0;
   AxisRun.Axis[5].Pos30.Speed := 0;
   AxisRun.Axis[5].Pos30.Reached := FALSE;
   AxisRun.Axis[6].Pos1.Position := 2.34;
   AxisRun.Axis[6].Pos1.Speed := 200;
   AxisRun.Axis[6].Pos1.Reached := FALSE;
   AxisRun.Axis[6].Pos2.Position := 76.0;
   AxisRun.Axis[6].Pos2.Speed := 200;
   AxisRun.Axis[6].Pos2.Reached := FALSE;
   AxisRun.Axis[6].Pos3.Position := 84.69;
   AxisRun.Axis[6].Pos3.Speed := 200;
   AxisRun.Axis[6].Pos3.Reached := FALSE;
   AxisRun.Axis[6].Pos4.Position := 84.69;
   AxisRun.Axis[6].Pos4.Speed := 200;
   AxisRun.Axis[6].Pos4.Reached := FALSE;
   AxisRun.Axis[6].Pos5.Position := 84.69;
   AxisRun.Axis[6].Pos5.Speed := 200;
   AxisRun.Axis[6].Pos5.Reached := FALSE;
   AxisRun.Axis[6].Pos6.Position := 84.69;
   AxisRun.Axis[6].Pos6.Speed := 200;
   AxisRun.Axis[6].Pos6.Reached := FALSE;
   AxisRun.Axis[6].Pos7.Position := 85.0;
   AxisRun.Axis[6].Pos7.Speed := 200;
   AxisRun.Axis[6].Pos7.Reached := FALSE;
   AxisRun.Axis[6].Pos8.Position := 88.53;
   AxisRun.Axis[6].Pos8.Speed := 200;
   AxisRun.Axis[6].Pos8.Reached := FALSE;
   AxisRun.Axis[6].Pos9.Position := 0.0;
   AxisRun.Axis[6].Pos9.Speed := 0;
   AxisRun.Axis[6].Pos9.Reached := FALSE;
   AxisRun.Axis[6].Pos10.Position := 0.0;
   AxisRun.Axis[6].Pos10.Speed := 0;
   AxisRun.Axis[6].Pos10.Reached := FALSE;
   AxisRun.Axis[6].Pos11.Position := 0.0;
   AxisRun.Axis[6].Pos11.Speed := 0;
   AxisRun.Axis[6].Pos11.Reached := FALSE;
   AxisRun.Axis[6].Pos12.Position := 0.0;
   AxisRun.Axis[6].Pos12.Speed := 0;
   AxisRun.Axis[6].Pos12.Reached := FALSE;
   AxisRun.Axis[6].Pos13.Position := 0.0;
   AxisRun.Axis[6].Pos13.Speed := 0;
   AxisRun.Axis[6].Pos13.Reached := FALSE;
   AxisRun.Axis[6].Pos14.Position := 0.0;
   AxisRun.Axis[6].Pos14.Speed := 0;
   AxisRun.Axis[6].Pos14.Reached := FALSE;
   AxisRun.Axis[6].Pos15.Position := 0.0;
   AxisRun.Axis[6].Pos15.Speed := 0;
   AxisRun.Axis[6].Pos15.Reached := FALSE;
   AxisRun.Axis[6].Pos16.Position := 0.0;
   AxisRun.Axis[6].Pos16.Speed := 0;
   AxisRun.Axis[6].Pos16.Reached := FALSE;
   AxisRun.Axis[6].Pos17.Position := 0.0;
   AxisRun.Axis[6].Pos17.Speed := 0;
   AxisRun.Axis[6].Pos17.Reached := FALSE;
   AxisRun.Axis[6].Pos18.Position := 0.0;
   AxisRun.Axis[6].Pos18.Speed := 0;
   AxisRun.Axis[6].Pos18.Reached := FALSE;
   AxisRun.Axis[6].Pos19.Position := 0.0;
   AxisRun.Axis[6].Pos19.Speed := 0;
   AxisRun.Axis[6].Pos19.Reached := FALSE;
   AxisRun.Axis[6].Pos20.Position := 0.0;
   AxisRun.Axis[6].Pos20.Speed := 0;
   AxisRun.Axis[6].Pos20.Reached := FALSE;
   AxisRun.Axis[6].Pos21.Position := 0.0;
   AxisRun.Axis[6].Pos21.Speed := 0;
   AxisRun.Axis[6].Pos21.Reached := FALSE;
   AxisRun.Axis[6].Pos22.Position := 0.0;
   AxisRun.Axis[6].Pos22.Speed := 0;
   AxisRun.Axis[6].Pos22.Reached := FALSE;
   AxisRun.Axis[6].Pos23.Position := 0.0;
   AxisRun.Axis[6].Pos23.Speed := 0;
   AxisRun.Axis[6].Pos23.Reached := FALSE;
   AxisRun.Axis[6].Pos24.Position := 0.0;
   AxisRun.Axis[6].Pos24.Speed := 0;
   AxisRun.Axis[6].Pos24.Reached := FALSE;
   AxisRun.Axis[6].Pos25.Position := 0.0;
   AxisRun.Axis[6].Pos25.Speed := 0;
   AxisRun.Axis[6].Pos25.Reached := FALSE;
   AxisRun.Axis[6].Pos26.Position := 0.0;
   AxisRun.Axis[6].Pos26.Speed := 0;
   AxisRun.Axis[6].Pos26.Reached := FALSE;
   AxisRun.Axis[6].Pos27.Position := 0.0;
   AxisRun.Axis[6].Pos27.Speed := 0;
   AxisRun.Axis[6].Pos27.Reached := FALSE;
   AxisRun.Axis[6].Pos28.Position := 0.0;
   AxisRun.Axis[6].Pos28.Speed := 0;
   AxisRun.Axis[6].Pos28.Reached := FALSE;
   AxisRun.Axis[6].Pos29.Position := 0.0;
   AxisRun.Axis[6].Pos29.Speed := 0;
   AxisRun.Axis[6].Pos29.Reached := FALSE;
   AxisRun.Axis[6].Pos30.Position := 0.0;
   AxisRun.Axis[6].Pos30.Speed := 0;
   AxisRun.Axis[6].Pos30.Reached := FALSE;
   AxisRun.Axis[7].Pos1.Position := 115.47;
   AxisRun.Axis[7].Pos1.Speed := 200;
   AxisRun.Axis[7].Pos1.Reached := FALSE;
   AxisRun.Axis[7].Pos2.Position := 115.47;
   AxisRun.Axis[7].Pos2.Speed := 200;
   AxisRun.Axis[7].Pos2.Reached := FALSE;
   AxisRun.Axis[7].Pos3.Position := 115.47;
   AxisRun.Axis[7].Pos3.Speed := 200;
   AxisRun.Axis[7].Pos3.Reached := FALSE;
   AxisRun.Axis[7].Pos4.Position := 115.47;
   AxisRun.Axis[7].Pos4.Speed := 200;
   AxisRun.Axis[7].Pos4.Reached := FALSE;
   AxisRun.Axis[7].Pos5.Position := 115.47;
   AxisRun.Axis[7].Pos5.Speed := 200;
   AxisRun.Axis[7].Pos5.Reached := FALSE;
   AxisRun.Axis[7].Pos6.Position := 110.18;
   AxisRun.Axis[7].Pos6.Speed := 200;
   AxisRun.Axis[7].Pos6.Reached := FALSE;
   AxisRun.Axis[7].Pos7.Position := 60.52;
   AxisRun.Axis[7].Pos7.Speed := 200;
   AxisRun.Axis[7].Pos7.Reached := FALSE;
   AxisRun.Axis[7].Pos8.Position := 80.0;
   AxisRun.Axis[7].Pos8.Speed := 100;
   AxisRun.Axis[7].Pos8.Reached := FALSE;
   AxisRun.Axis[7].Pos9.Position := 0.0;
   AxisRun.Axis[7].Pos9.Speed := 0;
   AxisRun.Axis[7].Pos9.Reached := FALSE;
   AxisRun.Axis[7].Pos10.Position := 0.0;
   AxisRun.Axis[7].Pos10.Speed := 0;
   AxisRun.Axis[7].Pos10.Reached := FALSE;
   AxisRun.Axis[7].Pos11.Position := 0.0;
   AxisRun.Axis[7].Pos11.Speed := 0;
   AxisRun.Axis[7].Pos11.Reached := FALSE;
   AxisRun.Axis[7].Pos12.Position := 0.0;
   AxisRun.Axis[7].Pos12.Speed := 0;
   AxisRun.Axis[7].Pos12.Reached := FALSE;
   AxisRun.Axis[7].Pos13.Position := 0.0;
   AxisRun.Axis[7].Pos13.Speed := 0;
   AxisRun.Axis[7].Pos13.Reached := FALSE;
   AxisRun.Axis[7].Pos14.Position := 0.0;
   AxisRun.Axis[7].Pos14.Speed := 0;
   AxisRun.Axis[7].Pos14.Reached := FALSE;
   AxisRun.Axis[7].Pos15.Position := 0.0;
   AxisRun.Axis[7].Pos15.Speed := 0;
   AxisRun.Axis[7].Pos15.Reached := FALSE;
   AxisRun.Axis[7].Pos16.Position := 0.0;
   AxisRun.Axis[7].Pos16.Speed := 0;
   AxisRun.Axis[7].Pos16.Reached := FALSE;
   AxisRun.Axis[7].Pos17.Position := 0.0;
   AxisRun.Axis[7].Pos17.Speed := 0;
   AxisRun.Axis[7].Pos17.Reached := FALSE;
   AxisRun.Axis[7].Pos18.Position := 0.0;
   AxisRun.Axis[7].Pos18.Speed := 0;
   AxisRun.Axis[7].Pos18.Reached := FALSE;
   AxisRun.Axis[7].Pos19.Position := 0.0;
   AxisRun.Axis[7].Pos19.Speed := 0;
   AxisRun.Axis[7].Pos19.Reached := FALSE;
   AxisRun.Axis[7].Pos20.Position := 0.0;
   AxisRun.Axis[7].Pos20.Speed := 0;
   AxisRun.Axis[7].Pos20.Reached := FALSE;
   AxisRun.Axis[7].Pos21.Position := 0.0;
   AxisRun.Axis[7].Pos21.Speed := 0;
   AxisRun.Axis[7].Pos21.Reached := FALSE;
   AxisRun.Axis[7].Pos22.Position := 0.0;
   AxisRun.Axis[7].Pos22.Speed := 0;
   AxisRun.Axis[7].Pos22.Reached := FALSE;
   AxisRun.Axis[7].Pos23.Position := 0.0;
   AxisRun.Axis[7].Pos23.Speed := 0;
   AxisRun.Axis[7].Pos23.Reached := FALSE;
   AxisRun.Axis[7].Pos24.Position := 0.0;
   AxisRun.Axis[7].Pos24.Speed := 0;
   AxisRun.Axis[7].Pos24.Reached := FALSE;
   AxisRun.Axis[7].Pos25.Position := 0.0;
   AxisRun.Axis[7].Pos25.Speed := 0;
   AxisRun.Axis[7].Pos25.Reached := FALSE;
   AxisRun.Axis[7].Pos26.Position := 0.0;
   AxisRun.Axis[7].Pos26.Speed := 0;
   AxisRun.Axis[7].Pos26.Reached := FALSE;
   AxisRun.Axis[7].Pos27.Position := 0.0;
   AxisRun.Axis[7].Pos27.Speed := 0;
   AxisRun.Axis[7].Pos27.Reached := FALSE;
   AxisRun.Axis[7].Pos28.Position := 0.0;
   AxisRun.Axis[7].Pos28.Speed := 0;
   AxisRun.Axis[7].Pos28.Reached := FALSE;
   AxisRun.Axis[7].Pos29.Position := 0.0;
   AxisRun.Axis[7].Pos29.Speed := 0;
   AxisRun.Axis[7].Pos29.Reached := FALSE;
   AxisRun.Axis[7].Pos30.Position := 0.0;
   AxisRun.Axis[7].Pos30.Speed := 0;
   AxisRun.Axis[7].Pos30.Reached := FALSE;
   AxisRun.Axis[8].Pos1.Position := 0.0;
   AxisRun.Axis[8].Pos1.Speed := 0;
   AxisRun.Axis[8].Pos1.Reached := FALSE;
   AxisRun.Axis[8].Pos2.Position := 0.0;
   AxisRun.Axis[8].Pos2.Speed := 0;
   AxisRun.Axis[8].Pos2.Reached := FALSE;
   AxisRun.Axis[8].Pos3.Position := 0.0;
   AxisRun.Axis[8].Pos3.Speed := 0;
   AxisRun.Axis[8].Pos3.Reached := FALSE;
   AxisRun.Axis[8].Pos4.Position := 0.0;
   AxisRun.Axis[8].Pos4.Speed := 0;
   AxisRun.Axis[8].Pos4.Reached := FALSE;
   AxisRun.Axis[8].Pos5.Position := 0.0;
   AxisRun.Axis[8].Pos5.Speed := 0;
   AxisRun.Axis[8].Pos5.Reached := FALSE;
   AxisRun.Axis[8].Pos6.Position := 0.0;
   AxisRun.Axis[8].Pos6.Speed := 0;
   AxisRun.Axis[8].Pos6.Reached := FALSE;
   AxisRun.Axis[8].Pos7.Position := 0.0;
   AxisRun.Axis[8].Pos7.Speed := 0;
   AxisRun.Axis[8].Pos7.Reached := FALSE;
   AxisRun.Axis[8].Pos8.Position := 0.0;
   AxisRun.Axis[8].Pos8.Speed := 0;
   AxisRun.Axis[8].Pos8.Reached := FALSE;
   AxisRun.Axis[8].Pos9.Position := 0.0;
   AxisRun.Axis[8].Pos9.Speed := 0;
   AxisRun.Axis[8].Pos9.Reached := FALSE;
   AxisRun.Axis[8].Pos10.Position := 0.0;
   AxisRun.Axis[8].Pos10.Speed := 0;
   AxisRun.Axis[8].Pos10.Reached := FALSE;
   AxisRun.Axis[8].Pos11.Position := 0.0;
   AxisRun.Axis[8].Pos11.Speed := 0;
   AxisRun.Axis[8].Pos11.Reached := FALSE;
   AxisRun.Axis[8].Pos12.Position := 0.0;
   AxisRun.Axis[8].Pos12.Speed := 0;
   AxisRun.Axis[8].Pos12.Reached := FALSE;
   AxisRun.Axis[8].Pos13.Position := 0.0;
   AxisRun.Axis[8].Pos13.Speed := 0;
   AxisRun.Axis[8].Pos13.Reached := FALSE;
   AxisRun.Axis[8].Pos14.Position := 0.0;
   AxisRun.Axis[8].Pos14.Speed := 0;
   AxisRun.Axis[8].Pos14.Reached := FALSE;
   AxisRun.Axis[8].Pos15.Position := 0.0;
   AxisRun.Axis[8].Pos15.Speed := 0;
   AxisRun.Axis[8].Pos15.Reached := FALSE;
   AxisRun.Axis[8].Pos16.Position := 0.0;
   AxisRun.Axis[8].Pos16.Speed := 0;
   AxisRun.Axis[8].Pos16.Reached := FALSE;
   AxisRun.Axis[8].Pos17.Position := 0.0;
   AxisRun.Axis[8].Pos17.Speed := 0;
   AxisRun.Axis[8].Pos17.Reached := FALSE;
   AxisRun.Axis[8].Pos18.Position := 0.0;
   AxisRun.Axis[8].Pos18.Speed := 0;
   AxisRun.Axis[8].Pos18.Reached := FALSE;
   AxisRun.Axis[8].Pos19.Position := 0.0;
   AxisRun.Axis[8].Pos19.Speed := 0;
   AxisRun.Axis[8].Pos19.Reached := FALSE;
   AxisRun.Axis[8].Pos20.Position := 0.0;
   AxisRun.Axis[8].Pos20.Speed := 0;
   AxisRun.Axis[8].Pos20.Reached := FALSE;
   AxisRun.Axis[8].Pos21.Position := 0.0;
   AxisRun.Axis[8].Pos21.Speed := 0;
   AxisRun.Axis[8].Pos21.Reached := FALSE;
   AxisRun.Axis[8].Pos22.Position := 0.0;
   AxisRun.Axis[8].Pos22.Speed := 0;
   AxisRun.Axis[8].Pos22.Reached := FALSE;
   AxisRun.Axis[8].Pos23.Position := 0.0;
   AxisRun.Axis[8].Pos23.Speed := 0;
   AxisRun.Axis[8].Pos23.Reached := FALSE;
   AxisRun.Axis[8].Pos24.Position := 0.0;
   AxisRun.Axis[8].Pos24.Speed := 0;
   AxisRun.Axis[8].Pos24.Reached := FALSE;
   AxisRun.Axis[8].Pos25.Position := 0.0;
   AxisRun.Axis[8].Pos25.Speed := 0;
   AxisRun.Axis[8].Pos25.Reached := FALSE;
   AxisRun.Axis[8].Pos26.Position := 0.0;
   AxisRun.Axis[8].Pos26.Speed := 0;
   AxisRun.Axis[8].Pos26.Reached := FALSE;
   AxisRun.Axis[8].Pos27.Position := 0.0;
   AxisRun.Axis[8].Pos27.Speed := 0;
   AxisRun.Axis[8].Pos27.Reached := FALSE;
   AxisRun.Axis[8].Pos28.Position := 0.0;
   AxisRun.Axis[8].Pos28.Speed := 0;
   AxisRun.Axis[8].Pos28.Reached := FALSE;
   AxisRun.Axis[8].Pos29.Position := 0.0;
   AxisRun.Axis[8].Pos29.Speed := 0;
   AxisRun.Axis[8].Pos29.Reached := FALSE;
   AxisRun.Axis[8].Pos30.Position := 0.0;
   AxisRun.Axis[8].Pos30.Speed := 0;
   AxisRun.Axis[8].Pos30.Reached := FALSE;
   AxisRun.Axis[9].Pos1.Position := 0.0;
   AxisRun.Axis[9].Pos1.Speed := 0;
   AxisRun.Axis[9].Pos1.Reached := FALSE;
   AxisRun.Axis[9].Pos2.Position := 0.0;
   AxisRun.Axis[9].Pos2.Speed := 0;
   AxisRun.Axis[9].Pos2.Reached := FALSE;
   AxisRun.Axis[9].Pos3.Position := 0.0;
   AxisRun.Axis[9].Pos3.Speed := 0;
   AxisRun.Axis[9].Pos3.Reached := FALSE;
   AxisRun.Axis[9].Pos4.Position := 0.0;
   AxisRun.Axis[9].Pos4.Speed := 0;
   AxisRun.Axis[9].Pos4.Reached := FALSE;
   AxisRun.Axis[9].Pos5.Position := 0.0;
   AxisRun.Axis[9].Pos5.Speed := 0;
   AxisRun.Axis[9].Pos5.Reached := FALSE;
   AxisRun.Axis[9].Pos6.Position := 0.0;
   AxisRun.Axis[9].Pos6.Speed := 0;
   AxisRun.Axis[9].Pos6.Reached := FALSE;
   AxisRun.Axis[9].Pos7.Position := 0.0;
   AxisRun.Axis[9].Pos7.Speed := 0;
   AxisRun.Axis[9].Pos7.Reached := FALSE;
   AxisRun.Axis[9].Pos8.Position := 0.0;
   AxisRun.Axis[9].Pos8.Speed := 0;
   AxisRun.Axis[9].Pos8.Reached := FALSE;
   AxisRun.Axis[9].Pos9.Position := 0.0;
   AxisRun.Axis[9].Pos9.Speed := 0;
   AxisRun.Axis[9].Pos9.Reached := FALSE;
   AxisRun.Axis[9].Pos10.Position := 0.0;
   AxisRun.Axis[9].Pos10.Speed := 0;
   AxisRun.Axis[9].Pos10.Reached := FALSE;
   AxisRun.Axis[9].Pos11.Position := 0.0;
   AxisRun.Axis[9].Pos11.Speed := 0;
   AxisRun.Axis[9].Pos11.Reached := FALSE;
   AxisRun.Axis[9].Pos12.Position := 0.0;
   AxisRun.Axis[9].Pos12.Speed := 0;
   AxisRun.Axis[9].Pos12.Reached := FALSE;
   AxisRun.Axis[9].Pos13.Position := 0.0;
   AxisRun.Axis[9].Pos13.Speed := 0;
   AxisRun.Axis[9].Pos13.Reached := FALSE;
   AxisRun.Axis[9].Pos14.Position := 0.0;
   AxisRun.Axis[9].Pos14.Speed := 0;
   AxisRun.Axis[9].Pos14.Reached := FALSE;
   AxisRun.Axis[9].Pos15.Position := 0.0;
   AxisRun.Axis[9].Pos15.Speed := 0;
   AxisRun.Axis[9].Pos15.Reached := FALSE;
   AxisRun.Axis[9].Pos16.Position := 0.0;
   AxisRun.Axis[9].Pos16.Speed := 0;
   AxisRun.Axis[9].Pos16.Reached := FALSE;
   AxisRun.Axis[9].Pos17.Position := 0.0;
   AxisRun.Axis[9].Pos17.Speed := 0;
   AxisRun.Axis[9].Pos17.Reached := FALSE;
   AxisRun.Axis[9].Pos18.Position := 0.0;
   AxisRun.Axis[9].Pos18.Speed := 0;
   AxisRun.Axis[9].Pos18.Reached := FALSE;
   AxisRun.Axis[9].Pos19.Position := 0.0;
   AxisRun.Axis[9].Pos19.Speed := 0;
   AxisRun.Axis[9].Pos19.Reached := FALSE;
   AxisRun.Axis[9].Pos20.Position := 0.0;
   AxisRun.Axis[9].Pos20.Speed := 0;
   AxisRun.Axis[9].Pos20.Reached := FALSE;
   AxisRun.Axis[9].Pos21.Position := 0.0;
   AxisRun.Axis[9].Pos21.Speed := 0;
   AxisRun.Axis[9].Pos21.Reached := FALSE;
   AxisRun.Axis[9].Pos22.Position := 0.0;
   AxisRun.Axis[9].Pos22.Speed := 0;
   AxisRun.Axis[9].Pos22.Reached := FALSE;
   AxisRun.Axis[9].Pos23.Position := 0.0;
   AxisRun.Axis[9].Pos23.Speed := 0;
   AxisRun.Axis[9].Pos23.Reached := FALSE;
   AxisRun.Axis[9].Pos24.Position := 0.0;
   AxisRun.Axis[9].Pos24.Speed := 0;
   AxisRun.Axis[9].Pos24.Reached := FALSE;
   AxisRun.Axis[9].Pos25.Position := 0.0;
   AxisRun.Axis[9].Pos25.Speed := 0;
   AxisRun.Axis[9].Pos25.Reached := FALSE;
   AxisRun.Axis[9].Pos26.Position := 0.0;
   AxisRun.Axis[9].Pos26.Speed := 0;
   AxisRun.Axis[9].Pos26.Reached := FALSE;
   AxisRun.Axis[9].Pos27.Position := 0.0;
   AxisRun.Axis[9].Pos27.Speed := 0;
   AxisRun.Axis[9].Pos27.Reached := FALSE;
   AxisRun.Axis[9].Pos28.Position := 0.0;
   AxisRun.Axis[9].Pos28.Speed := 0;
   AxisRun.Axis[9].Pos28.Reached := FALSE;
   AxisRun.Axis[9].Pos29.Position := 0.0;
   AxisRun.Axis[9].Pos29.Speed := 0;
   AxisRun.Axis[9].Pos29.Reached := FALSE;
   AxisRun.Axis[9].Pos30.Position := 0.0;
   AxisRun.Axis[9].Pos30.Speed := 0;
   AxisRun.Axis[9].Pos30.Reached := FALSE;
   AxisRun.Axis[10].Pos1.Position := 0.0;
   AxisRun.Axis[10].Pos1.Speed := 0;
   AxisRun.Axis[10].Pos1.Reached := FALSE;
   AxisRun.Axis[10].Pos2.Position := 0.0;
   AxisRun.Axis[10].Pos2.Speed := 0;
   AxisRun.Axis[10].Pos2.Reached := FALSE;
   AxisRun.Axis[10].Pos3.Position := 0.0;
   AxisRun.Axis[10].Pos3.Speed := 0;
   AxisRun.Axis[10].Pos3.Reached := FALSE;
   AxisRun.Axis[10].Pos4.Position := 0.0;
   AxisRun.Axis[10].Pos4.Speed := 0;
   AxisRun.Axis[10].Pos4.Reached := FALSE;
   AxisRun.Axis[10].Pos5.Position := 0.0;
   AxisRun.Axis[10].Pos5.Speed := 0;
   AxisRun.Axis[10].Pos5.Reached := FALSE;
   AxisRun.Axis[10].Pos6.Position := 0.0;
   AxisRun.Axis[10].Pos6.Speed := 0;
   AxisRun.Axis[10].Pos6.Reached := FALSE;
   AxisRun.Axis[10].Pos7.Position := 0.0;
   AxisRun.Axis[10].Pos7.Speed := 0;
   AxisRun.Axis[10].Pos7.Reached := FALSE;
   AxisRun.Axis[10].Pos8.Position := 0.0;
   AxisRun.Axis[10].Pos8.Speed := 0;
   AxisRun.Axis[10].Pos8.Reached := FALSE;
   AxisRun.Axis[10].Pos9.Position := 0.0;
   AxisRun.Axis[10].Pos9.Speed := 0;
   AxisRun.Axis[10].Pos9.Reached := FALSE;
   AxisRun.Axis[10].Pos10.Position := 0.0;
   AxisRun.Axis[10].Pos10.Speed := 0;
   AxisRun.Axis[10].Pos10.Reached := FALSE;
   AxisRun.Axis[10].Pos11.Position := 0.0;
   AxisRun.Axis[10].Pos11.Speed := 0;
   AxisRun.Axis[10].Pos11.Reached := FALSE;
   AxisRun.Axis[10].Pos12.Position := 0.0;
   AxisRun.Axis[10].Pos12.Speed := 0;
   AxisRun.Axis[10].Pos12.Reached := FALSE;
   AxisRun.Axis[10].Pos13.Position := 0.0;
   AxisRun.Axis[10].Pos13.Speed := 0;
   AxisRun.Axis[10].Pos13.Reached := FALSE;
   AxisRun.Axis[10].Pos14.Position := 0.0;
   AxisRun.Axis[10].Pos14.Speed := 0;
   AxisRun.Axis[10].Pos14.Reached := FALSE;
   AxisRun.Axis[10].Pos15.Position := 0.0;
   AxisRun.Axis[10].Pos15.Speed := 0;
   AxisRun.Axis[10].Pos15.Reached := FALSE;
   AxisRun.Axis[10].Pos16.Position := 0.0;
   AxisRun.Axis[10].Pos16.Speed := 0;
   AxisRun.Axis[10].Pos16.Reached := FALSE;
   AxisRun.Axis[10].Pos17.Position := 0.0;
   AxisRun.Axis[10].Pos17.Speed := 0;
   AxisRun.Axis[10].Pos17.Reached := FALSE;
   AxisRun.Axis[10].Pos18.Position := 0.0;
   AxisRun.Axis[10].Pos18.Speed := 0;
   AxisRun.Axis[10].Pos18.Reached := FALSE;
   AxisRun.Axis[10].Pos19.Position := 0.0;
   AxisRun.Axis[10].Pos19.Speed := 0;
   AxisRun.Axis[10].Pos19.Reached := FALSE;
   AxisRun.Axis[10].Pos20.Position := 0.0;
   AxisRun.Axis[10].Pos20.Speed := 0;
   AxisRun.Axis[10].Pos20.Reached := FALSE;
   AxisRun.Axis[10].Pos21.Position := 0.0;
   AxisRun.Axis[10].Pos21.Speed := 0;
   AxisRun.Axis[10].Pos21.Reached := FALSE;
   AxisRun.Axis[10].Pos22.Position := 0.0;
   AxisRun.Axis[10].Pos22.Speed := 0;
   AxisRun.Axis[10].Pos22.Reached := FALSE;
   AxisRun.Axis[10].Pos23.Position := 0.0;
   AxisRun.Axis[10].Pos23.Speed := 0;
   AxisRun.Axis[10].Pos23.Reached := FALSE;
   AxisRun.Axis[10].Pos24.Position := 0.0;
   AxisRun.Axis[10].Pos24.Speed := 0;
   AxisRun.Axis[10].Pos24.Reached := FALSE;
   AxisRun.Axis[10].Pos25.Position := 0.0;
   AxisRun.Axis[10].Pos25.Speed := 0;
   AxisRun.Axis[10].Pos25.Reached := FALSE;
   AxisRun.Axis[10].Pos26.Position := 0.0;
   AxisRun.Axis[10].Pos26.Speed := 0;
   AxisRun.Axis[10].Pos26.Reached := FALSE;
   AxisRun.Axis[10].Pos27.Position := 0.0;
   AxisRun.Axis[10].Pos27.Speed := 0;
   AxisRun.Axis[10].Pos27.Reached := FALSE;
   AxisRun.Axis[10].Pos28.Position := 0.0;
   AxisRun.Axis[10].Pos28.Speed := 0;
   AxisRun.Axis[10].Pos28.Reached := FALSE;
   AxisRun.Axis[10].Pos29.Position := 0.0;
   AxisRun.Axis[10].Pos29.Speed := 0;
   AxisRun.Axis[10].Pos29.Reached := FALSE;
   AxisRun.Axis[10].Pos30.Position := 0.0;
   AxisRun.Axis[10].Pos30.Speed := 0;
   AxisRun.Axis[10].Pos30.Reached := FALSE;
   AxisRun.Axis[11].Pos1.Position := 0.0;
   AxisRun.Axis[11].Pos1.Speed := 0;
   AxisRun.Axis[11].Pos1.Reached := FALSE;
   AxisRun.Axis[11].Pos2.Position := 0.0;
   AxisRun.Axis[11].Pos2.Speed := 0;
   AxisRun.Axis[11].Pos2.Reached := FALSE;
   AxisRun.Axis[11].Pos3.Position := 0.0;
   AxisRun.Axis[11].Pos3.Speed := 0;
   AxisRun.Axis[11].Pos3.Reached := FALSE;
   AxisRun.Axis[11].Pos4.Position := 0.0;
   AxisRun.Axis[11].Pos4.Speed := 0;
   AxisRun.Axis[11].Pos4.Reached := FALSE;
   AxisRun.Axis[11].Pos5.Position := 0.0;
   AxisRun.Axis[11].Pos5.Speed := 0;
   AxisRun.Axis[11].Pos5.Reached := FALSE;
   AxisRun.Axis[11].Pos6.Position := 0.0;
   AxisRun.Axis[11].Pos6.Speed := 0;
   AxisRun.Axis[11].Pos6.Reached := FALSE;
   AxisRun.Axis[11].Pos7.Position := 0.0;
   AxisRun.Axis[11].Pos7.Speed := 0;
   AxisRun.Axis[11].Pos7.Reached := FALSE;
   AxisRun.Axis[11].Pos8.Position := 0.0;
   AxisRun.Axis[11].Pos8.Speed := 0;
   AxisRun.Axis[11].Pos8.Reached := FALSE;
   AxisRun.Axis[11].Pos9.Position := 0.0;
   AxisRun.Axis[11].Pos9.Speed := 0;
   AxisRun.Axis[11].Pos9.Reached := FALSE;
   AxisRun.Axis[11].Pos10.Position := 0.0;
   AxisRun.Axis[11].Pos10.Speed := 0;
   AxisRun.Axis[11].Pos10.Reached := FALSE;
   AxisRun.Axis[11].Pos11.Position := 0.0;
   AxisRun.Axis[11].Pos11.Speed := 0;
   AxisRun.Axis[11].Pos11.Reached := FALSE;
   AxisRun.Axis[11].Pos12.Position := 0.0;
   AxisRun.Axis[11].Pos12.Speed := 0;
   AxisRun.Axis[11].Pos12.Reached := FALSE;
   AxisRun.Axis[11].Pos13.Position := 0.0;
   AxisRun.Axis[11].Pos13.Speed := 0;
   AxisRun.Axis[11].Pos13.Reached := FALSE;
   AxisRun.Axis[11].Pos14.Position := 0.0;
   AxisRun.Axis[11].Pos14.Speed := 0;
   AxisRun.Axis[11].Pos14.Reached := FALSE;
   AxisRun.Axis[11].Pos15.Position := 0.0;
   AxisRun.Axis[11].Pos15.Speed := 0;
   AxisRun.Axis[11].Pos15.Reached := FALSE;
   AxisRun.Axis[11].Pos16.Position := 0.0;
   AxisRun.Axis[11].Pos16.Speed := 0;
   AxisRun.Axis[11].Pos16.Reached := FALSE;
   AxisRun.Axis[11].Pos17.Position := 0.0;
   AxisRun.Axis[11].Pos17.Speed := 0;
   AxisRun.Axis[11].Pos17.Reached := FALSE;
   AxisRun.Axis[11].Pos18.Position := 0.0;
   AxisRun.Axis[11].Pos18.Speed := 0;
   AxisRun.Axis[11].Pos18.Reached := FALSE;
   AxisRun.Axis[11].Pos19.Position := 0.0;
   AxisRun.Axis[11].Pos19.Speed := 0;
   AxisRun.Axis[11].Pos19.Reached := FALSE;
   AxisRun.Axis[11].Pos20.Position := 0.0;
   AxisRun.Axis[11].Pos20.Speed := 0;
   AxisRun.Axis[11].Pos20.Reached := FALSE;
   AxisRun.Axis[11].Pos21.Position := 0.0;
   AxisRun.Axis[11].Pos21.Speed := 0;
   AxisRun.Axis[11].Pos21.Reached := FALSE;
   AxisRun.Axis[11].Pos22.Position := 0.0;
   AxisRun.Axis[11].Pos22.Speed := 0;
   AxisRun.Axis[11].Pos22.Reached := FALSE;
   AxisRun.Axis[11].Pos23.Position := 0.0;
   AxisRun.Axis[11].Pos23.Speed := 0;
   AxisRun.Axis[11].Pos23.Reached := FALSE;
   AxisRun.Axis[11].Pos24.Position := 0.0;
   AxisRun.Axis[11].Pos24.Speed := 0;
   AxisRun.Axis[11].Pos24.Reached := FALSE;
   AxisRun.Axis[11].Pos25.Position := 0.0;
   AxisRun.Axis[11].Pos25.Speed := 0;
   AxisRun.Axis[11].Pos25.Reached := FALSE;
   AxisRun.Axis[11].Pos26.Position := 0.0;
   AxisRun.Axis[11].Pos26.Speed := 0;
   AxisRun.Axis[11].Pos26.Reached := FALSE;
   AxisRun.Axis[11].Pos27.Position := 0.0;
   AxisRun.Axis[11].Pos27.Speed := 0;
   AxisRun.Axis[11].Pos27.Reached := FALSE;
   AxisRun.Axis[11].Pos28.Position := 0.0;
   AxisRun.Axis[11].Pos28.Speed := 0;
   AxisRun.Axis[11].Pos28.Reached := FALSE;
   AxisRun.Axis[11].Pos29.Position := 0.0;
   AxisRun.Axis[11].Pos29.Speed := 0;
   AxisRun.Axis[11].Pos29.Reached := FALSE;
   AxisRun.Axis[11].Pos30.Position := 0.0;
   AxisRun.Axis[11].Pos30.Speed := 0;
   AxisRun.Axis[11].Pos30.Reached := FALSE;
   AxisRun.Axis[12].Pos1.Position := 0.0;
   AxisRun.Axis[12].Pos1.Speed := 0;
   AxisRun.Axis[12].Pos1.Reached := FALSE;
   AxisRun.Axis[12].Pos2.Position := 0.0;
   AxisRun.Axis[12].Pos2.Speed := 0;
   AxisRun.Axis[12].Pos2.Reached := FALSE;
   AxisRun.Axis[12].Pos3.Position := 0.0;
   AxisRun.Axis[12].Pos3.Speed := 0;
   AxisRun.Axis[12].Pos3.Reached := FALSE;
   AxisRun.Axis[12].Pos4.Position := 0.0;
   AxisRun.Axis[12].Pos4.Speed := 0;
   AxisRun.Axis[12].Pos4.Reached := FALSE;
   AxisRun.Axis[12].Pos5.Position := 0.0;
   AxisRun.Axis[12].Pos5.Speed := 0;
   AxisRun.Axis[12].Pos5.Reached := FALSE;
   AxisRun.Axis[12].Pos6.Position := 0.0;
   AxisRun.Axis[12].Pos6.Speed := 0;
   AxisRun.Axis[12].Pos6.Reached := FALSE;
   AxisRun.Axis[12].Pos7.Position := 0.0;
   AxisRun.Axis[12].Pos7.Speed := 0;
   AxisRun.Axis[12].Pos7.Reached := FALSE;
   AxisRun.Axis[12].Pos8.Position := 0.0;
   AxisRun.Axis[12].Pos8.Speed := 0;
   AxisRun.Axis[12].Pos8.Reached := FALSE;
   AxisRun.Axis[12].Pos9.Position := 0.0;
   AxisRun.Axis[12].Pos9.Speed := 0;
   AxisRun.Axis[12].Pos9.Reached := FALSE;
   AxisRun.Axis[12].Pos10.Position := 0.0;
   AxisRun.Axis[12].Pos10.Speed := 0;
   AxisRun.Axis[12].Pos10.Reached := FALSE;
   AxisRun.Axis[12].Pos11.Position := 0.0;
   AxisRun.Axis[12].Pos11.Speed := 0;
   AxisRun.Axis[12].Pos11.Reached := FALSE;
   AxisRun.Axis[12].Pos12.Position := 0.0;
   AxisRun.Axis[12].Pos12.Speed := 0;
   AxisRun.Axis[12].Pos12.Reached := FALSE;
   AxisRun.Axis[12].Pos13.Position := 0.0;
   AxisRun.Axis[12].Pos13.Speed := 0;
   AxisRun.Axis[12].Pos13.Reached := FALSE;
   AxisRun.Axis[12].Pos14.Position := 0.0;
   AxisRun.Axis[12].Pos14.Speed := 0;
   AxisRun.Axis[12].Pos14.Reached := FALSE;
   AxisRun.Axis[12].Pos15.Position := 0.0;
   AxisRun.Axis[12].Pos15.Speed := 0;
   AxisRun.Axis[12].Pos15.Reached := FALSE;
   AxisRun.Axis[12].Pos16.Position := 0.0;
   AxisRun.Axis[12].Pos16.Speed := 0;
   AxisRun.Axis[12].Pos16.Reached := FALSE;
   AxisRun.Axis[12].Pos17.Position := 0.0;
   AxisRun.Axis[12].Pos17.Speed := 0;
   AxisRun.Axis[12].Pos17.Reached := FALSE;
   AxisRun.Axis[12].Pos18.Position := 0.0;
   AxisRun.Axis[12].Pos18.Speed := 0;
   AxisRun.Axis[12].Pos18.Reached := FALSE;
   AxisRun.Axis[12].Pos19.Position := 0.0;
   AxisRun.Axis[12].Pos19.Speed := 0;
   AxisRun.Axis[12].Pos19.Reached := FALSE;
   AxisRun.Axis[12].Pos20.Position := 0.0;
   AxisRun.Axis[12].Pos20.Speed := 0;
   AxisRun.Axis[12].Pos20.Reached := FALSE;
   AxisRun.Axis[12].Pos21.Position := 0.0;
   AxisRun.Axis[12].Pos21.Speed := 0;
   AxisRun.Axis[12].Pos21.Reached := FALSE;
   AxisRun.Axis[12].Pos22.Position := 0.0;
   AxisRun.Axis[12].Pos22.Speed := 0;
   AxisRun.Axis[12].Pos22.Reached := FALSE;
   AxisRun.Axis[12].Pos23.Position := 0.0;
   AxisRun.Axis[12].Pos23.Speed := 0;
   AxisRun.Axis[12].Pos23.Reached := FALSE;
   AxisRun.Axis[12].Pos24.Position := 0.0;
   AxisRun.Axis[12].Pos24.Speed := 0;
   AxisRun.Axis[12].Pos24.Reached := FALSE;
   AxisRun.Axis[12].Pos25.Position := 0.0;
   AxisRun.Axis[12].Pos25.Speed := 0;
   AxisRun.Axis[12].Pos25.Reached := FALSE;
   AxisRun.Axis[12].Pos26.Position := 0.0;
   AxisRun.Axis[12].Pos26.Speed := 0;
   AxisRun.Axis[12].Pos26.Reached := FALSE;
   AxisRun.Axis[12].Pos27.Position := 0.0;
   AxisRun.Axis[12].Pos27.Speed := 0;
   AxisRun.Axis[12].Pos27.Reached := FALSE;
   AxisRun.Axis[12].Pos28.Position := 0.0;
   AxisRun.Axis[12].Pos28.Speed := 0;
   AxisRun.Axis[12].Pos28.Reached := FALSE;
   AxisRun.Axis[12].Pos29.Position := 0.0;
   AxisRun.Axis[12].Pos29.Speed := 0;
   AxisRun.Axis[12].Pos29.Reached := FALSE;
   AxisRun.Axis[12].Pos30.Position := 0.0;
   AxisRun.Axis[12].Pos30.Speed := 0;
   AxisRun.Axis[12].Pos30.Reached := FALSE;
   AxisRun.Axis[13].Pos1.Position := 0.0;
   AxisRun.Axis[13].Pos1.Speed := 0;
   AxisRun.Axis[13].Pos1.Reached := FALSE;
   AxisRun.Axis[13].Pos2.Position := 0.0;
   AxisRun.Axis[13].Pos2.Speed := 0;
   AxisRun.Axis[13].Pos2.Reached := FALSE;
   AxisRun.Axis[13].Pos3.Position := 0.0;
   AxisRun.Axis[13].Pos3.Speed := 0;
   AxisRun.Axis[13].Pos3.Reached := FALSE;
   AxisRun.Axis[13].Pos4.Position := 0.0;
   AxisRun.Axis[13].Pos4.Speed := 0;
   AxisRun.Axis[13].Pos4.Reached := FALSE;
   AxisRun.Axis[13].Pos5.Position := 0.0;
   AxisRun.Axis[13].Pos5.Speed := 0;
   AxisRun.Axis[13].Pos5.Reached := FALSE;
   AxisRun.Axis[13].Pos6.Position := 0.0;
   AxisRun.Axis[13].Pos6.Speed := 0;
   AxisRun.Axis[13].Pos6.Reached := FALSE;
   AxisRun.Axis[13].Pos7.Position := 0.0;
   AxisRun.Axis[13].Pos7.Speed := 0;
   AxisRun.Axis[13].Pos7.Reached := FALSE;
   AxisRun.Axis[13].Pos8.Position := 0.0;
   AxisRun.Axis[13].Pos8.Speed := 0;
   AxisRun.Axis[13].Pos8.Reached := FALSE;
   AxisRun.Axis[13].Pos9.Position := 0.0;
   AxisRun.Axis[13].Pos9.Speed := 0;
   AxisRun.Axis[13].Pos9.Reached := FALSE;
   AxisRun.Axis[13].Pos10.Position := 0.0;
   AxisRun.Axis[13].Pos10.Speed := 0;
   AxisRun.Axis[13].Pos10.Reached := FALSE;
   AxisRun.Axis[13].Pos11.Position := 0.0;
   AxisRun.Axis[13].Pos11.Speed := 0;
   AxisRun.Axis[13].Pos11.Reached := FALSE;
   AxisRun.Axis[13].Pos12.Position := 0.0;
   AxisRun.Axis[13].Pos12.Speed := 0;
   AxisRun.Axis[13].Pos12.Reached := FALSE;
   AxisRun.Axis[13].Pos13.Position := 0.0;
   AxisRun.Axis[13].Pos13.Speed := 0;
   AxisRun.Axis[13].Pos13.Reached := FALSE;
   AxisRun.Axis[13].Pos14.Position := 0.0;
   AxisRun.Axis[13].Pos14.Speed := 0;
   AxisRun.Axis[13].Pos14.Reached := FALSE;
   AxisRun.Axis[13].Pos15.Position := 0.0;
   AxisRun.Axis[13].Pos15.Speed := 0;
   AxisRun.Axis[13].Pos15.Reached := FALSE;
   AxisRun.Axis[13].Pos16.Position := 0.0;
   AxisRun.Axis[13].Pos16.Speed := 0;
   AxisRun.Axis[13].Pos16.Reached := FALSE;
   AxisRun.Axis[13].Pos17.Position := 0.0;
   AxisRun.Axis[13].Pos17.Speed := 0;
   AxisRun.Axis[13].Pos17.Reached := FALSE;
   AxisRun.Axis[13].Pos18.Position := 0.0;
   AxisRun.Axis[13].Pos18.Speed := 0;
   AxisRun.Axis[13].Pos18.Reached := FALSE;
   AxisRun.Axis[13].Pos19.Position := 0.0;
   AxisRun.Axis[13].Pos19.Speed := 0;
   AxisRun.Axis[13].Pos19.Reached := FALSE;
   AxisRun.Axis[13].Pos20.Position := 0.0;
   AxisRun.Axis[13].Pos20.Speed := 0;
   AxisRun.Axis[13].Pos20.Reached := FALSE;
   AxisRun.Axis[13].Pos21.Position := 0.0;
   AxisRun.Axis[13].Pos21.Speed := 0;
   AxisRun.Axis[13].Pos21.Reached := FALSE;
   AxisRun.Axis[13].Pos22.Position := 0.0;
   AxisRun.Axis[13].Pos22.Speed := 0;
   AxisRun.Axis[13].Pos22.Reached := FALSE;
   AxisRun.Axis[13].Pos23.Position := 0.0;
   AxisRun.Axis[13].Pos23.Speed := 0;
   AxisRun.Axis[13].Pos23.Reached := FALSE;
   AxisRun.Axis[13].Pos24.Position := 0.0;
   AxisRun.Axis[13].Pos24.Speed := 0;
   AxisRun.Axis[13].Pos24.Reached := FALSE;
   AxisRun.Axis[13].Pos25.Position := 0.0;
   AxisRun.Axis[13].Pos25.Speed := 0;
   AxisRun.Axis[13].Pos25.Reached := FALSE;
   AxisRun.Axis[13].Pos26.Position := 0.0;
   AxisRun.Axis[13].Pos26.Speed := 0;
   AxisRun.Axis[13].Pos26.Reached := FALSE;
   AxisRun.Axis[13].Pos27.Position := 0.0;
   AxisRun.Axis[13].Pos27.Speed := 0;
   AxisRun.Axis[13].Pos27.Reached := FALSE;
   AxisRun.Axis[13].Pos28.Position := 0.0;
   AxisRun.Axis[13].Pos28.Speed := 0;
   AxisRun.Axis[13].Pos28.Reached := FALSE;
   AxisRun.Axis[13].Pos29.Position := 0.0;
   AxisRun.Axis[13].Pos29.Speed := 0;
   AxisRun.Axis[13].Pos29.Reached := FALSE;
   AxisRun.Axis[13].Pos30.Position := 0.0;
   AxisRun.Axis[13].Pos30.Speed := 0;
   AxisRun.Axis[13].Pos30.Reached := FALSE;
   AxisRun.Axis[14].Pos1.Position := 0.0;
   AxisRun.Axis[14].Pos1.Speed := 0;
   AxisRun.Axis[14].Pos1.Reached := FALSE;
   AxisRun.Axis[14].Pos2.Position := 0.0;
   AxisRun.Axis[14].Pos2.Speed := 0;
   AxisRun.Axis[14].Pos2.Reached := FALSE;
   AxisRun.Axis[14].Pos3.Position := 0.0;
   AxisRun.Axis[14].Pos3.Speed := 0;
   AxisRun.Axis[14].Pos3.Reached := FALSE;
   AxisRun.Axis[14].Pos4.Position := 0.0;
   AxisRun.Axis[14].Pos4.Speed := 0;
   AxisRun.Axis[14].Pos4.Reached := FALSE;
   AxisRun.Axis[14].Pos5.Position := 0.0;
   AxisRun.Axis[14].Pos5.Speed := 0;
   AxisRun.Axis[14].Pos5.Reached := FALSE;
   AxisRun.Axis[14].Pos6.Position := 0.0;
   AxisRun.Axis[14].Pos6.Speed := 0;
   AxisRun.Axis[14].Pos6.Reached := FALSE;
   AxisRun.Axis[14].Pos7.Position := 0.0;
   AxisRun.Axis[14].Pos7.Speed := 0;
   AxisRun.Axis[14].Pos7.Reached := FALSE;
   AxisRun.Axis[14].Pos8.Position := 0.0;
   AxisRun.Axis[14].Pos8.Speed := 0;
   AxisRun.Axis[14].Pos8.Reached := FALSE;
   AxisRun.Axis[14].Pos9.Position := 0.0;
   AxisRun.Axis[14].Pos9.Speed := 0;
   AxisRun.Axis[14].Pos9.Reached := FALSE;
   AxisRun.Axis[14].Pos10.Position := 0.0;
   AxisRun.Axis[14].Pos10.Speed := 0;
   AxisRun.Axis[14].Pos10.Reached := FALSE;
   AxisRun.Axis[14].Pos11.Position := 0.0;
   AxisRun.Axis[14].Pos11.Speed := 0;
   AxisRun.Axis[14].Pos11.Reached := FALSE;
   AxisRun.Axis[14].Pos12.Position := 0.0;
   AxisRun.Axis[14].Pos12.Speed := 0;
   AxisRun.Axis[14].Pos12.Reached := FALSE;
   AxisRun.Axis[14].Pos13.Position := 0.0;
   AxisRun.Axis[14].Pos13.Speed := 0;
   AxisRun.Axis[14].Pos13.Reached := FALSE;
   AxisRun.Axis[14].Pos14.Position := 0.0;
   AxisRun.Axis[14].Pos14.Speed := 0;
   AxisRun.Axis[14].Pos14.Reached := FALSE;
   AxisRun.Axis[14].Pos15.Position := 0.0;
   AxisRun.Axis[14].Pos15.Speed := 0;
   AxisRun.Axis[14].Pos15.Reached := FALSE;
   AxisRun.Axis[14].Pos16.Position := 0.0;
   AxisRun.Axis[14].Pos16.Speed := 0;
   AxisRun.Axis[14].Pos16.Reached := FALSE;
   AxisRun.Axis[14].Pos17.Position := 0.0;
   AxisRun.Axis[14].Pos17.Speed := 0;
   AxisRun.Axis[14].Pos17.Reached := FALSE;
   AxisRun.Axis[14].Pos18.Position := 0.0;
   AxisRun.Axis[14].Pos18.Speed := 0;
   AxisRun.Axis[14].Pos18.Reached := FALSE;
   AxisRun.Axis[14].Pos19.Position := 0.0;
   AxisRun.Axis[14].Pos19.Speed := 0;
   AxisRun.Axis[14].Pos19.Reached := FALSE;
   AxisRun.Axis[14].Pos20.Position := 0.0;
   AxisRun.Axis[14].Pos20.Speed := 0;
   AxisRun.Axis[14].Pos20.Reached := FALSE;
   AxisRun.Axis[14].Pos21.Position := 0.0;
   AxisRun.Axis[14].Pos21.Speed := 0;
   AxisRun.Axis[14].Pos21.Reached := FALSE;
   AxisRun.Axis[14].Pos22.Position := 0.0;
   AxisRun.Axis[14].Pos22.Speed := 0;
   AxisRun.Axis[14].Pos22.Reached := FALSE;
   AxisRun.Axis[14].Pos23.Position := 0.0;
   AxisRun.Axis[14].Pos23.Speed := 0;
   AxisRun.Axis[14].Pos23.Reached := FALSE;
   AxisRun.Axis[14].Pos24.Position := 0.0;
   AxisRun.Axis[14].Pos24.Speed := 0;
   AxisRun.Axis[14].Pos24.Reached := FALSE;
   AxisRun.Axis[14].Pos25.Position := 0.0;
   AxisRun.Axis[14].Pos25.Speed := 0;
   AxisRun.Axis[14].Pos25.Reached := FALSE;
   AxisRun.Axis[14].Pos26.Position := 0.0;
   AxisRun.Axis[14].Pos26.Speed := 0;
   AxisRun.Axis[14].Pos26.Reached := FALSE;
   AxisRun.Axis[14].Pos27.Position := 0.0;
   AxisRun.Axis[14].Pos27.Speed := 0;
   AxisRun.Axis[14].Pos27.Reached := FALSE;
   AxisRun.Axis[14].Pos28.Position := 0.0;
   AxisRun.Axis[14].Pos28.Speed := 0;
   AxisRun.Axis[14].Pos28.Reached := FALSE;
   AxisRun.Axis[14].Pos29.Position := 0.0;
   AxisRun.Axis[14].Pos29.Speed := 0;
   AxisRun.Axis[14].Pos29.Reached := FALSE;
   AxisRun.Axis[14].Pos30.Position := 0.0;
   AxisRun.Axis[14].Pos30.Speed := 0;
   AxisRun.Axis[14].Pos30.Reached := FALSE;
   AxisRun.Axis[15].Pos1.Position := 0.0;
   AxisRun.Axis[15].Pos1.Speed := 0;
   AxisRun.Axis[15].Pos1.Reached := FALSE;
   AxisRun.Axis[15].Pos2.Position := 0.0;
   AxisRun.Axis[15].Pos2.Speed := 0;
   AxisRun.Axis[15].Pos2.Reached := FALSE;
   AxisRun.Axis[15].Pos3.Position := 0.0;
   AxisRun.Axis[15].Pos3.Speed := 0;
   AxisRun.Axis[15].Pos3.Reached := FALSE;
   AxisRun.Axis[15].Pos4.Position := 0.0;
   AxisRun.Axis[15].Pos4.Speed := 0;
   AxisRun.Axis[15].Pos4.Reached := FALSE;
   AxisRun.Axis[15].Pos5.Position := 0.0;
   AxisRun.Axis[15].Pos5.Speed := 0;
   AxisRun.Axis[15].Pos5.Reached := FALSE;
   AxisRun.Axis[15].Pos6.Position := 0.0;
   AxisRun.Axis[15].Pos6.Speed := 0;
   AxisRun.Axis[15].Pos6.Reached := FALSE;
   AxisRun.Axis[15].Pos7.Position := 0.0;
   AxisRun.Axis[15].Pos7.Speed := 0;
   AxisRun.Axis[15].Pos7.Reached := FALSE;
   AxisRun.Axis[15].Pos8.Position := 0.0;
   AxisRun.Axis[15].Pos8.Speed := 0;
   AxisRun.Axis[15].Pos8.Reached := FALSE;
   AxisRun.Axis[15].Pos9.Position := 0.0;
   AxisRun.Axis[15].Pos9.Speed := 0;
   AxisRun.Axis[15].Pos9.Reached := FALSE;
   AxisRun.Axis[15].Pos10.Position := 0.0;
   AxisRun.Axis[15].Pos10.Speed := 0;
   AxisRun.Axis[15].Pos10.Reached := FALSE;
   AxisRun.Axis[15].Pos11.Position := 0.0;
   AxisRun.Axis[15].Pos11.Speed := 0;
   AxisRun.Axis[15].Pos11.Reached := FALSE;
   AxisRun.Axis[15].Pos12.Position := 0.0;
   AxisRun.Axis[15].Pos12.Speed := 0;
   AxisRun.Axis[15].Pos12.Reached := FALSE;
   AxisRun.Axis[15].Pos13.Position := 0.0;
   AxisRun.Axis[15].Pos13.Speed := 0;
   AxisRun.Axis[15].Pos13.Reached := FALSE;
   AxisRun.Axis[15].Pos14.Position := 0.0;
   AxisRun.Axis[15].Pos14.Speed := 0;
   AxisRun.Axis[15].Pos14.Reached := FALSE;
   AxisRun.Axis[15].Pos15.Position := 0.0;
   AxisRun.Axis[15].Pos15.Speed := 0;
   AxisRun.Axis[15].Pos15.Reached := FALSE;
   AxisRun.Axis[15].Pos16.Position := 0.0;
   AxisRun.Axis[15].Pos16.Speed := 0;
   AxisRun.Axis[15].Pos16.Reached := FALSE;
   AxisRun.Axis[15].Pos17.Position := 0.0;
   AxisRun.Axis[15].Pos17.Speed := 0;
   AxisRun.Axis[15].Pos17.Reached := FALSE;
   AxisRun.Axis[15].Pos18.Position := 0.0;
   AxisRun.Axis[15].Pos18.Speed := 0;
   AxisRun.Axis[15].Pos18.Reached := FALSE;
   AxisRun.Axis[15].Pos19.Position := 0.0;
   AxisRun.Axis[15].Pos19.Speed := 0;
   AxisRun.Axis[15].Pos19.Reached := FALSE;
   AxisRun.Axis[15].Pos20.Position := 0.0;
   AxisRun.Axis[15].Pos20.Speed := 0;
   AxisRun.Axis[15].Pos20.Reached := FALSE;
   AxisRun.Axis[15].Pos21.Position := 0.0;
   AxisRun.Axis[15].Pos21.Speed := 0;
   AxisRun.Axis[15].Pos21.Reached := FALSE;
   AxisRun.Axis[15].Pos22.Position := 0.0;
   AxisRun.Axis[15].Pos22.Speed := 0;
   AxisRun.Axis[15].Pos22.Reached := FALSE;
   AxisRun.Axis[15].Pos23.Position := 0.0;
   AxisRun.Axis[15].Pos23.Speed := 0;
   AxisRun.Axis[15].Pos23.Reached := FALSE;
   AxisRun.Axis[15].Pos24.Position := 0.0;
   AxisRun.Axis[15].Pos24.Speed := 0;
   AxisRun.Axis[15].Pos24.Reached := FALSE;
   AxisRun.Axis[15].Pos25.Position := 0.0;
   AxisRun.Axis[15].Pos25.Speed := 0;
   AxisRun.Axis[15].Pos25.Reached := FALSE;
   AxisRun.Axis[15].Pos26.Position := 0.0;
   AxisRun.Axis[15].Pos26.Speed := 0;
   AxisRun.Axis[15].Pos26.Reached := FALSE;
   AxisRun.Axis[15].Pos27.Position := 0.0;
   AxisRun.Axis[15].Pos27.Speed := 0;
   AxisRun.Axis[15].Pos27.Reached := FALSE;
   AxisRun.Axis[15].Pos28.Position := 0.0;
   AxisRun.Axis[15].Pos28.Speed := 0;
   AxisRun.Axis[15].Pos28.Reached := FALSE;
   AxisRun.Axis[15].Pos29.Position := 0.0;
   AxisRun.Axis[15].Pos29.Speed := 0;
   AxisRun.Axis[15].Pos29.Reached := FALSE;
   AxisRun.Axis[15].Pos30.Position := 0.0;
   AxisRun.Axis[15].Pos30.Speed := 0;
   AxisRun.Axis[15].Pos30.Reached := FALSE;
   AxisNuw.Axis[1].Pos1.Position := 0.0;
   AxisNuw.Axis[1].Pos1.Speed := 0;
   AxisNuw.Axis[1].Pos1.Reached := FALSE;
   AxisNuw.Axis[1].Pos2.Position := 0.0;
   AxisNuw.Axis[1].Pos2.Speed := 0;
   AxisNuw.Axis[1].Pos2.Reached := FALSE;
   AxisNuw.Axis[1].Pos3.Position := 0.0;
   AxisNuw.Axis[1].Pos3.Speed := 0;
   AxisNuw.Axis[1].Pos3.Reached := FALSE;
   AxisNuw.Axis[1].Pos4.Position := 0.0;
   AxisNuw.Axis[1].Pos4.Speed := 0;
   AxisNuw.Axis[1].Pos4.Reached := FALSE;
   AxisNuw.Axis[1].Pos5.Position := 0.0;
   AxisNuw.Axis[1].Pos5.Speed := 0;
   AxisNuw.Axis[1].Pos5.Reached := FALSE;
   AxisNuw.Axis[1].Pos6.Position := 0.0;
   AxisNuw.Axis[1].Pos6.Speed := 0;
   AxisNuw.Axis[1].Pos6.Reached := FALSE;
   AxisNuw.Axis[1].Pos7.Position := 0.0;
   AxisNuw.Axis[1].Pos7.Speed := 0;
   AxisNuw.Axis[1].Pos7.Reached := FALSE;
   AxisNuw.Axis[1].Pos8.Position := 0.0;
   AxisNuw.Axis[1].Pos8.Speed := 0;
   AxisNuw.Axis[1].Pos8.Reached := FALSE;
   AxisNuw.Axis[1].Pos9.Position := 0.0;
   AxisNuw.Axis[1].Pos9.Speed := 0;
   AxisNuw.Axis[1].Pos9.Reached := FALSE;
   AxisNuw.Axis[1].Pos10.Position := 0.0;
   AxisNuw.Axis[1].Pos10.Speed := 0;
   AxisNuw.Axis[1].Pos10.Reached := FALSE;
   AxisNuw.Axis[1].Pos11.Position := 0.0;
   AxisNuw.Axis[1].Pos11.Speed := 0;
   AxisNuw.Axis[1].Pos11.Reached := FALSE;
   AxisNuw.Axis[1].Pos12.Position := 0.0;
   AxisNuw.Axis[1].Pos12.Speed := 0;
   AxisNuw.Axis[1].Pos12.Reached := FALSE;
   AxisNuw.Axis[1].Pos13.Position := 0.0;
   AxisNuw.Axis[1].Pos13.Speed := 0;
   AxisNuw.Axis[1].Pos13.Reached := FALSE;
   AxisNuw.Axis[1].Pos14.Position := 0.0;
   AxisNuw.Axis[1].Pos14.Speed := 0;
   AxisNuw.Axis[1].Pos14.Reached := FALSE;
   AxisNuw.Axis[1].Pos15.Position := 0.0;
   AxisNuw.Axis[1].Pos15.Speed := 0;
   AxisNuw.Axis[1].Pos15.Reached := FALSE;
   AxisNuw.Axis[1].Pos16.Position := 0.0;
   AxisNuw.Axis[1].Pos16.Speed := 0;
   AxisNuw.Axis[1].Pos16.Reached := FALSE;
   AxisNuw.Axis[1].Pos17.Position := 0.0;
   AxisNuw.Axis[1].Pos17.Speed := 0;
   AxisNuw.Axis[1].Pos17.Reached := FALSE;
   AxisNuw.Axis[1].Pos18.Position := 0.0;
   AxisNuw.Axis[1].Pos18.Speed := 0;
   AxisNuw.Axis[1].Pos18.Reached := FALSE;
   AxisNuw.Axis[1].Pos19.Position := 0.0;
   AxisNuw.Axis[1].Pos19.Speed := 0;
   AxisNuw.Axis[1].Pos19.Reached := FALSE;
   AxisNuw.Axis[1].Pos20.Position := 0.0;
   AxisNuw.Axis[1].Pos20.Speed := 0;
   AxisNuw.Axis[1].Pos20.Reached := FALSE;
   AxisNuw.Axis[1].Pos21.Position := 0.0;
   AxisNuw.Axis[1].Pos21.Speed := 0;
   AxisNuw.Axis[1].Pos21.Reached := FALSE;
   AxisNuw.Axis[1].Pos22.Position := 0.0;
   AxisNuw.Axis[1].Pos22.Speed := 0;
   AxisNuw.Axis[1].Pos22.Reached := FALSE;
   AxisNuw.Axis[1].Pos23.Position := 0.0;
   AxisNuw.Axis[1].Pos23.Speed := 0;
   AxisNuw.Axis[1].Pos23.Reached := FALSE;
   AxisNuw.Axis[1].Pos24.Position := 0.0;
   AxisNuw.Axis[1].Pos24.Speed := 0;
   AxisNuw.Axis[1].Pos24.Reached := FALSE;
   AxisNuw.Axis[1].Pos25.Position := 0.0;
   AxisNuw.Axis[1].Pos25.Speed := 0;
   AxisNuw.Axis[1].Pos25.Reached := FALSE;
   AxisNuw.Axis[1].Pos26.Position := 0.0;
   AxisNuw.Axis[1].Pos26.Speed := 0;
   AxisNuw.Axis[1].Pos26.Reached := FALSE;
   AxisNuw.Axis[1].Pos27.Position := 0.0;
   AxisNuw.Axis[1].Pos27.Speed := 0;
   AxisNuw.Axis[1].Pos27.Reached := FALSE;
   AxisNuw.Axis[1].Pos28.Position := 0.0;
   AxisNuw.Axis[1].Pos28.Speed := 0;
   AxisNuw.Axis[1].Pos28.Reached := FALSE;
   AxisNuw.Axis[1].Pos29.Position := 0.0;
   AxisNuw.Axis[1].Pos29.Speed := 0;
   AxisNuw.Axis[1].Pos29.Reached := FALSE;
   AxisNuw.Axis[1].Pos30.Position := 0.0;
   AxisNuw.Axis[1].Pos30.Speed := 0;
   AxisNuw.Axis[1].Pos30.Reached := FALSE;
   AxisNuw.Axis[2].Pos1.Position := 0.0;
   AxisNuw.Axis[2].Pos1.Speed := 0;
   AxisNuw.Axis[2].Pos1.Reached := FALSE;
   AxisNuw.Axis[2].Pos2.Position := 0.0;
   AxisNuw.Axis[2].Pos2.Speed := 0;
   AxisNuw.Axis[2].Pos2.Reached := FALSE;
   AxisNuw.Axis[2].Pos3.Position := 0.0;
   AxisNuw.Axis[2].Pos3.Speed := 0;
   AxisNuw.Axis[2].Pos3.Reached := FALSE;
   AxisNuw.Axis[2].Pos4.Position := 0.0;
   AxisNuw.Axis[2].Pos4.Speed := 0;
   AxisNuw.Axis[2].Pos4.Reached := FALSE;
   AxisNuw.Axis[2].Pos5.Position := 0.0;
   AxisNuw.Axis[2].Pos5.Speed := 0;
   AxisNuw.Axis[2].Pos5.Reached := FALSE;
   AxisNuw.Axis[2].Pos6.Position := 0.0;
   AxisNuw.Axis[2].Pos6.Speed := 0;
   AxisNuw.Axis[2].Pos6.Reached := FALSE;
   AxisNuw.Axis[2].Pos7.Position := 0.0;
   AxisNuw.Axis[2].Pos7.Speed := 0;
   AxisNuw.Axis[2].Pos7.Reached := FALSE;
   AxisNuw.Axis[2].Pos8.Position := 0.0;
   AxisNuw.Axis[2].Pos8.Speed := 0;
   AxisNuw.Axis[2].Pos8.Reached := FALSE;
   AxisNuw.Axis[2].Pos9.Position := 0.0;
   AxisNuw.Axis[2].Pos9.Speed := 0;
   AxisNuw.Axis[2].Pos9.Reached := FALSE;
   AxisNuw.Axis[2].Pos10.Position := 0.0;
   AxisNuw.Axis[2].Pos10.Speed := 0;
   AxisNuw.Axis[2].Pos10.Reached := FALSE;
   AxisNuw.Axis[2].Pos11.Position := 0.0;
   AxisNuw.Axis[2].Pos11.Speed := 0;
   AxisNuw.Axis[2].Pos11.Reached := FALSE;
   AxisNuw.Axis[2].Pos12.Position := 0.0;
   AxisNuw.Axis[2].Pos12.Speed := 0;
   AxisNuw.Axis[2].Pos12.Reached := FALSE;
   AxisNuw.Axis[2].Pos13.Position := 0.0;
   AxisNuw.Axis[2].Pos13.Speed := 0;
   AxisNuw.Axis[2].Pos13.Reached := FALSE;
   AxisNuw.Axis[2].Pos14.Position := 0.0;
   AxisNuw.Axis[2].Pos14.Speed := 0;
   AxisNuw.Axis[2].Pos14.Reached := FALSE;
   AxisNuw.Axis[2].Pos15.Position := 0.0;
   AxisNuw.Axis[2].Pos15.Speed := 0;
   AxisNuw.Axis[2].Pos15.Reached := FALSE;
   AxisNuw.Axis[2].Pos16.Position := 0.0;
   AxisNuw.Axis[2].Pos16.Speed := 0;
   AxisNuw.Axis[2].Pos16.Reached := FALSE;
   AxisNuw.Axis[2].Pos17.Position := 0.0;
   AxisNuw.Axis[2].Pos17.Speed := 0;
   AxisNuw.Axis[2].Pos17.Reached := FALSE;
   AxisNuw.Axis[2].Pos18.Position := 0.0;
   AxisNuw.Axis[2].Pos18.Speed := 0;
   AxisNuw.Axis[2].Pos18.Reached := FALSE;
   AxisNuw.Axis[2].Pos19.Position := 0.0;
   AxisNuw.Axis[2].Pos19.Speed := 0;
   AxisNuw.Axis[2].Pos19.Reached := FALSE;
   AxisNuw.Axis[2].Pos20.Position := 0.0;
   AxisNuw.Axis[2].Pos20.Speed := 0;
   AxisNuw.Axis[2].Pos20.Reached := FALSE;
   AxisNuw.Axis[2].Pos21.Position := 0.0;
   AxisNuw.Axis[2].Pos21.Speed := 0;
   AxisNuw.Axis[2].Pos21.Reached := FALSE;
   AxisNuw.Axis[2].Pos22.Position := 0.0;
   AxisNuw.Axis[2].Pos22.Speed := 0;
   AxisNuw.Axis[2].Pos22.Reached := FALSE;
   AxisNuw.Axis[2].Pos23.Position := 0.0;
   AxisNuw.Axis[2].Pos23.Speed := 0;
   AxisNuw.Axis[2].Pos23.Reached := FALSE;
   AxisNuw.Axis[2].Pos24.Position := 0.0;
   AxisNuw.Axis[2].Pos24.Speed := 0;
   AxisNuw.Axis[2].Pos24.Reached := FALSE;
   AxisNuw.Axis[2].Pos25.Position := 0.0;
   AxisNuw.Axis[2].Pos25.Speed := 0;
   AxisNuw.Axis[2].Pos25.Reached := FALSE;
   AxisNuw.Axis[2].Pos26.Position := 0.0;
   AxisNuw.Axis[2].Pos26.Speed := 0;
   AxisNuw.Axis[2].Pos26.Reached := FALSE;
   AxisNuw.Axis[2].Pos27.Position := 0.0;
   AxisNuw.Axis[2].Pos27.Speed := 0;
   AxisNuw.Axis[2].Pos27.Reached := FALSE;
   AxisNuw.Axis[2].Pos28.Position := 0.0;
   AxisNuw.Axis[2].Pos28.Speed := 0;
   AxisNuw.Axis[2].Pos28.Reached := FALSE;
   AxisNuw.Axis[2].Pos29.Position := 0.0;
   AxisNuw.Axis[2].Pos29.Speed := 0;
   AxisNuw.Axis[2].Pos29.Reached := FALSE;
   AxisNuw.Axis[2].Pos30.Position := 0.0;
   AxisNuw.Axis[2].Pos30.Speed := 0;
   AxisNuw.Axis[2].Pos30.Reached := FALSE;
   AxisNuw.Axis[3].Pos1.Position := 0.0;
   AxisNuw.Axis[3].Pos1.Speed := 0;
   AxisNuw.Axis[3].Pos1.Reached := FALSE;
   AxisNuw.Axis[3].Pos2.Position := 0.0;
   AxisNuw.Axis[3].Pos2.Speed := 0;
   AxisNuw.Axis[3].Pos2.Reached := FALSE;
   AxisNuw.Axis[3].Pos3.Position := 0.0;
   AxisNuw.Axis[3].Pos3.Speed := 0;
   AxisNuw.Axis[3].Pos3.Reached := FALSE;
   AxisNuw.Axis[3].Pos4.Position := 0.0;
   AxisNuw.Axis[3].Pos4.Speed := 0;
   AxisNuw.Axis[3].Pos4.Reached := FALSE;
   AxisNuw.Axis[3].Pos5.Position := 0.0;
   AxisNuw.Axis[3].Pos5.Speed := 0;
   AxisNuw.Axis[3].Pos5.Reached := FALSE;
   AxisNuw.Axis[3].Pos6.Position := 0.0;
   AxisNuw.Axis[3].Pos6.Speed := 0;
   AxisNuw.Axis[3].Pos6.Reached := FALSE;
   AxisNuw.Axis[3].Pos7.Position := 0.0;
   AxisNuw.Axis[3].Pos7.Speed := 0;
   AxisNuw.Axis[3].Pos7.Reached := FALSE;
   AxisNuw.Axis[3].Pos8.Position := 0.0;
   AxisNuw.Axis[3].Pos8.Speed := 0;
   AxisNuw.Axis[3].Pos8.Reached := FALSE;
   AxisNuw.Axis[3].Pos9.Position := 0.0;
   AxisNuw.Axis[3].Pos9.Speed := 0;
   AxisNuw.Axis[3].Pos9.Reached := FALSE;
   AxisNuw.Axis[3].Pos10.Position := 0.0;
   AxisNuw.Axis[3].Pos10.Speed := 0;
   AxisNuw.Axis[3].Pos10.Reached := FALSE;
   AxisNuw.Axis[3].Pos11.Position := 0.0;
   AxisNuw.Axis[3].Pos11.Speed := 0;
   AxisNuw.Axis[3].Pos11.Reached := FALSE;
   AxisNuw.Axis[3].Pos12.Position := 0.0;
   AxisNuw.Axis[3].Pos12.Speed := 0;
   AxisNuw.Axis[3].Pos12.Reached := FALSE;
   AxisNuw.Axis[3].Pos13.Position := 0.0;
   AxisNuw.Axis[3].Pos13.Speed := 0;
   AxisNuw.Axis[3].Pos13.Reached := FALSE;
   AxisNuw.Axis[3].Pos14.Position := 0.0;
   AxisNuw.Axis[3].Pos14.Speed := 0;
   AxisNuw.Axis[3].Pos14.Reached := FALSE;
   AxisNuw.Axis[3].Pos15.Position := 0.0;
   AxisNuw.Axis[3].Pos15.Speed := 0;
   AxisNuw.Axis[3].Pos15.Reached := FALSE;
   AxisNuw.Axis[3].Pos16.Position := 0.0;
   AxisNuw.Axis[3].Pos16.Speed := 0;
   AxisNuw.Axis[3].Pos16.Reached := FALSE;
   AxisNuw.Axis[3].Pos17.Position := 0.0;
   AxisNuw.Axis[3].Pos17.Speed := 0;
   AxisNuw.Axis[3].Pos17.Reached := FALSE;
   AxisNuw.Axis[3].Pos18.Position := 0.0;
   AxisNuw.Axis[3].Pos18.Speed := 0;
   AxisNuw.Axis[3].Pos18.Reached := FALSE;
   AxisNuw.Axis[3].Pos19.Position := 0.0;
   AxisNuw.Axis[3].Pos19.Speed := 0;
   AxisNuw.Axis[3].Pos19.Reached := FALSE;
   AxisNuw.Axis[3].Pos20.Position := 0.0;
   AxisNuw.Axis[3].Pos20.Speed := 0;
   AxisNuw.Axis[3].Pos20.Reached := FALSE;
   AxisNuw.Axis[3].Pos21.Position := 0.0;
   AxisNuw.Axis[3].Pos21.Speed := 0;
   AxisNuw.Axis[3].Pos21.Reached := FALSE;
   AxisNuw.Axis[3].Pos22.Position := 0.0;
   AxisNuw.Axis[3].Pos22.Speed := 0;
   AxisNuw.Axis[3].Pos22.Reached := FALSE;
   AxisNuw.Axis[3].Pos23.Position := 0.0;
   AxisNuw.Axis[3].Pos23.Speed := 0;
   AxisNuw.Axis[3].Pos23.Reached := FALSE;
   AxisNuw.Axis[3].Pos24.Position := 0.0;
   AxisNuw.Axis[3].Pos24.Speed := 0;
   AxisNuw.Axis[3].Pos24.Reached := FALSE;
   AxisNuw.Axis[3].Pos25.Position := 0.0;
   AxisNuw.Axis[3].Pos25.Speed := 0;
   AxisNuw.Axis[3].Pos25.Reached := FALSE;
   AxisNuw.Axis[3].Pos26.Position := 0.0;
   AxisNuw.Axis[3].Pos26.Speed := 0;
   AxisNuw.Axis[3].Pos26.Reached := FALSE;
   AxisNuw.Axis[3].Pos27.Position := 0.0;
   AxisNuw.Axis[3].Pos27.Speed := 0;
   AxisNuw.Axis[3].Pos27.Reached := FALSE;
   AxisNuw.Axis[3].Pos28.Position := 0.0;
   AxisNuw.Axis[3].Pos28.Speed := 0;
   AxisNuw.Axis[3].Pos28.Reached := FALSE;
   AxisNuw.Axis[3].Pos29.Position := 0.0;
   AxisNuw.Axis[3].Pos29.Speed := 0;
   AxisNuw.Axis[3].Pos29.Reached := FALSE;
   AxisNuw.Axis[3].Pos30.Position := 0.0;
   AxisNuw.Axis[3].Pos30.Speed := 0;
   AxisNuw.Axis[3].Pos30.Reached := FALSE;
   AxisNuw.Axis[4].Pos1.Position := 0.0;
   AxisNuw.Axis[4].Pos1.Speed := 0;
   AxisNuw.Axis[4].Pos1.Reached := FALSE;
   AxisNuw.Axis[4].Pos2.Position := 0.0;
   AxisNuw.Axis[4].Pos2.Speed := 0;
   AxisNuw.Axis[4].Pos2.Reached := FALSE;
   AxisNuw.Axis[4].Pos3.Position := 0.0;
   AxisNuw.Axis[4].Pos3.Speed := 0;
   AxisNuw.Axis[4].Pos3.Reached := FALSE;
   AxisNuw.Axis[4].Pos4.Position := 0.0;
   AxisNuw.Axis[4].Pos4.Speed := 0;
   AxisNuw.Axis[4].Pos4.Reached := FALSE;
   AxisNuw.Axis[4].Pos5.Position := 0.0;
   AxisNuw.Axis[4].Pos5.Speed := 0;
   AxisNuw.Axis[4].Pos5.Reached := FALSE;
   AxisNuw.Axis[4].Pos6.Position := 0.0;
   AxisNuw.Axis[4].Pos6.Speed := 0;
   AxisNuw.Axis[4].Pos6.Reached := FALSE;
   AxisNuw.Axis[4].Pos7.Position := 0.0;
   AxisNuw.Axis[4].Pos7.Speed := 0;
   AxisNuw.Axis[4].Pos7.Reached := FALSE;
   AxisNuw.Axis[4].Pos8.Position := 0.0;
   AxisNuw.Axis[4].Pos8.Speed := 0;
   AxisNuw.Axis[4].Pos8.Reached := FALSE;
   AxisNuw.Axis[4].Pos9.Position := 0.0;
   AxisNuw.Axis[4].Pos9.Speed := 0;
   AxisNuw.Axis[4].Pos9.Reached := FALSE;
   AxisNuw.Axis[4].Pos10.Position := 0.0;
   AxisNuw.Axis[4].Pos10.Speed := 0;
   AxisNuw.Axis[4].Pos10.Reached := FALSE;
   AxisNuw.Axis[4].Pos11.Position := 0.0;
   AxisNuw.Axis[4].Pos11.Speed := 0;
   AxisNuw.Axis[4].Pos11.Reached := FALSE;
   AxisNuw.Axis[4].Pos12.Position := 0.0;
   AxisNuw.Axis[4].Pos12.Speed := 0;
   AxisNuw.Axis[4].Pos12.Reached := FALSE;
   AxisNuw.Axis[4].Pos13.Position := 0.0;
   AxisNuw.Axis[4].Pos13.Speed := 0;
   AxisNuw.Axis[4].Pos13.Reached := FALSE;
   AxisNuw.Axis[4].Pos14.Position := 0.0;
   AxisNuw.Axis[4].Pos14.Speed := 0;
   AxisNuw.Axis[4].Pos14.Reached := FALSE;
   AxisNuw.Axis[4].Pos15.Position := 0.0;
   AxisNuw.Axis[4].Pos15.Speed := 0;
   AxisNuw.Axis[4].Pos15.Reached := FALSE;
   AxisNuw.Axis[4].Pos16.Position := 0.0;
   AxisNuw.Axis[4].Pos16.Speed := 0;
   AxisNuw.Axis[4].Pos16.Reached := FALSE;
   AxisNuw.Axis[4].Pos17.Position := 0.0;
   AxisNuw.Axis[4].Pos17.Speed := 0;
   AxisNuw.Axis[4].Pos17.Reached := FALSE;
   AxisNuw.Axis[4].Pos18.Position := 0.0;
   AxisNuw.Axis[4].Pos18.Speed := 0;
   AxisNuw.Axis[4].Pos18.Reached := FALSE;
   AxisNuw.Axis[4].Pos19.Position := 0.0;
   AxisNuw.Axis[4].Pos19.Speed := 0;
   AxisNuw.Axis[4].Pos19.Reached := FALSE;
   AxisNuw.Axis[4].Pos20.Position := 0.0;
   AxisNuw.Axis[4].Pos20.Speed := 0;
   AxisNuw.Axis[4].Pos20.Reached := FALSE;
   AxisNuw.Axis[4].Pos21.Position := 0.0;
   AxisNuw.Axis[4].Pos21.Speed := 0;
   AxisNuw.Axis[4].Pos21.Reached := FALSE;
   AxisNuw.Axis[4].Pos22.Position := 0.0;
   AxisNuw.Axis[4].Pos22.Speed := 0;
   AxisNuw.Axis[4].Pos22.Reached := FALSE;
   AxisNuw.Axis[4].Pos23.Position := 0.0;
   AxisNuw.Axis[4].Pos23.Speed := 0;
   AxisNuw.Axis[4].Pos23.Reached := FALSE;
   AxisNuw.Axis[4].Pos24.Position := 0.0;
   AxisNuw.Axis[4].Pos24.Speed := 0;
   AxisNuw.Axis[4].Pos24.Reached := FALSE;
   AxisNuw.Axis[4].Pos25.Position := 0.0;
   AxisNuw.Axis[4].Pos25.Speed := 0;
   AxisNuw.Axis[4].Pos25.Reached := FALSE;
   AxisNuw.Axis[4].Pos26.Position := 0.0;
   AxisNuw.Axis[4].Pos26.Speed := 0;
   AxisNuw.Axis[4].Pos26.Reached := FALSE;
   AxisNuw.Axis[4].Pos27.Position := 0.0;
   AxisNuw.Axis[4].Pos27.Speed := 0;
   AxisNuw.Axis[4].Pos27.Reached := FALSE;
   AxisNuw.Axis[4].Pos28.Position := 0.0;
   AxisNuw.Axis[4].Pos28.Speed := 0;
   AxisNuw.Axis[4].Pos28.Reached := FALSE;
   AxisNuw.Axis[4].Pos29.Position := 0.0;
   AxisNuw.Axis[4].Pos29.Speed := 0;
   AxisNuw.Axis[4].Pos29.Reached := FALSE;
   AxisNuw.Axis[4].Pos30.Position := 0.0;
   AxisNuw.Axis[4].Pos30.Speed := 0;
   AxisNuw.Axis[4].Pos30.Reached := FALSE;
   AxisNuw.Axis[5].Pos1.Position := 0.0;
   AxisNuw.Axis[5].Pos1.Speed := 0;
   AxisNuw.Axis[5].Pos1.Reached := FALSE;
   AxisNuw.Axis[5].Pos2.Position := 0.0;
   AxisNuw.Axis[5].Pos2.Speed := 0;
   AxisNuw.Axis[5].Pos2.Reached := FALSE;
   AxisNuw.Axis[5].Pos3.Position := 0.0;
   AxisNuw.Axis[5].Pos3.Speed := 0;
   AxisNuw.Axis[5].Pos3.Reached := FALSE;
   AxisNuw.Axis[5].Pos4.Position := 0.0;
   AxisNuw.Axis[5].Pos4.Speed := 0;
   AxisNuw.Axis[5].Pos4.Reached := FALSE;
   AxisNuw.Axis[5].Pos5.Position := 0.0;
   AxisNuw.Axis[5].Pos5.Speed := 0;
   AxisNuw.Axis[5].Pos5.Reached := FALSE;
   AxisNuw.Axis[5].Pos6.Position := 0.0;
   AxisNuw.Axis[5].Pos6.Speed := 0;
   AxisNuw.Axis[5].Pos6.Reached := FALSE;
   AxisNuw.Axis[5].Pos7.Position := 0.0;
   AxisNuw.Axis[5].Pos7.Speed := 0;
   AxisNuw.Axis[5].Pos7.Reached := FALSE;
   AxisNuw.Axis[5].Pos8.Position := 0.0;
   AxisNuw.Axis[5].Pos8.Speed := 0;
   AxisNuw.Axis[5].Pos8.Reached := FALSE;
   AxisNuw.Axis[5].Pos9.Position := 0.0;
   AxisNuw.Axis[5].Pos9.Speed := 0;
   AxisNuw.Axis[5].Pos9.Reached := FALSE;
   AxisNuw.Axis[5].Pos10.Position := 0.0;
   AxisNuw.Axis[5].Pos10.Speed := 0;
   AxisNuw.Axis[5].Pos10.Reached := FALSE;
   AxisNuw.Axis[5].Pos11.Position := 0.0;
   AxisNuw.Axis[5].Pos11.Speed := 0;
   AxisNuw.Axis[5].Pos11.Reached := FALSE;
   AxisNuw.Axis[5].Pos12.Position := 0.0;
   AxisNuw.Axis[5].Pos12.Speed := 0;
   AxisNuw.Axis[5].Pos12.Reached := FALSE;
   AxisNuw.Axis[5].Pos13.Position := 0.0;
   AxisNuw.Axis[5].Pos13.Speed := 0;
   AxisNuw.Axis[5].Pos13.Reached := FALSE;
   AxisNuw.Axis[5].Pos14.Position := 0.0;
   AxisNuw.Axis[5].Pos14.Speed := 0;
   AxisNuw.Axis[5].Pos14.Reached := FALSE;
   AxisNuw.Axis[5].Pos15.Position := 0.0;
   AxisNuw.Axis[5].Pos15.Speed := 0;
   AxisNuw.Axis[5].Pos15.Reached := FALSE;
   AxisNuw.Axis[5].Pos16.Position := 0.0;
   AxisNuw.Axis[5].Pos16.Speed := 0;
   AxisNuw.Axis[5].Pos16.Reached := FALSE;
   AxisNuw.Axis[5].Pos17.Position := 0.0;
   AxisNuw.Axis[5].Pos17.Speed := 0;
   AxisNuw.Axis[5].Pos17.Reached := FALSE;
   AxisNuw.Axis[5].Pos18.Position := 0.0;
   AxisNuw.Axis[5].Pos18.Speed := 0;
   AxisNuw.Axis[5].Pos18.Reached := FALSE;
   AxisNuw.Axis[5].Pos19.Position := 0.0;
   AxisNuw.Axis[5].Pos19.Speed := 0;
   AxisNuw.Axis[5].Pos19.Reached := FALSE;
   AxisNuw.Axis[5].Pos20.Position := 0.0;
   AxisNuw.Axis[5].Pos20.Speed := 0;
   AxisNuw.Axis[5].Pos20.Reached := FALSE;
   AxisNuw.Axis[5].Pos21.Position := 0.0;
   AxisNuw.Axis[5].Pos21.Speed := 0;
   AxisNuw.Axis[5].Pos21.Reached := FALSE;
   AxisNuw.Axis[5].Pos22.Position := 0.0;
   AxisNuw.Axis[5].Pos22.Speed := 0;
   AxisNuw.Axis[5].Pos22.Reached := FALSE;
   AxisNuw.Axis[5].Pos23.Position := 0.0;
   AxisNuw.Axis[5].Pos23.Speed := 0;
   AxisNuw.Axis[5].Pos23.Reached := FALSE;
   AxisNuw.Axis[5].Pos24.Position := 0.0;
   AxisNuw.Axis[5].Pos24.Speed := 0;
   AxisNuw.Axis[5].Pos24.Reached := FALSE;
   AxisNuw.Axis[5].Pos25.Position := 0.0;
   AxisNuw.Axis[5].Pos25.Speed := 0;
   AxisNuw.Axis[5].Pos25.Reached := FALSE;
   AxisNuw.Axis[5].Pos26.Position := 0.0;
   AxisNuw.Axis[5].Pos26.Speed := 0;
   AxisNuw.Axis[5].Pos26.Reached := FALSE;
   AxisNuw.Axis[5].Pos27.Position := 0.0;
   AxisNuw.Axis[5].Pos27.Speed := 0;
   AxisNuw.Axis[5].Pos27.Reached := FALSE;
   AxisNuw.Axis[5].Pos28.Position := 0.0;
   AxisNuw.Axis[5].Pos28.Speed := 0;
   AxisNuw.Axis[5].Pos28.Reached := FALSE;
   AxisNuw.Axis[5].Pos29.Position := 0.0;
   AxisNuw.Axis[5].Pos29.Speed := 0;
   AxisNuw.Axis[5].Pos29.Reached := FALSE;
   AxisNuw.Axis[5].Pos30.Position := 0.0;
   AxisNuw.Axis[5].Pos30.Speed := 0;
   AxisNuw.Axis[5].Pos30.Reached := FALSE;
   AxisNuw.Axis[6].Pos1.Position := 0.0;
   AxisNuw.Axis[6].Pos1.Speed := 0;
   AxisNuw.Axis[6].Pos1.Reached := FALSE;
   AxisNuw.Axis[6].Pos2.Position := 0.0;
   AxisNuw.Axis[6].Pos2.Speed := 0;
   AxisNuw.Axis[6].Pos2.Reached := FALSE;
   AxisNuw.Axis[6].Pos3.Position := 0.0;
   AxisNuw.Axis[6].Pos3.Speed := 0;
   AxisNuw.Axis[6].Pos3.Reached := FALSE;
   AxisNuw.Axis[6].Pos4.Position := 0.0;
   AxisNuw.Axis[6].Pos4.Speed := 0;
   AxisNuw.Axis[6].Pos4.Reached := FALSE;
   AxisNuw.Axis[6].Pos5.Position := 0.0;
   AxisNuw.Axis[6].Pos5.Speed := 0;
   AxisNuw.Axis[6].Pos5.Reached := FALSE;
   AxisNuw.Axis[6].Pos6.Position := 0.0;
   AxisNuw.Axis[6].Pos6.Speed := 0;
   AxisNuw.Axis[6].Pos6.Reached := FALSE;
   AxisNuw.Axis[6].Pos7.Position := 0.0;
   AxisNuw.Axis[6].Pos7.Speed := 0;
   AxisNuw.Axis[6].Pos7.Reached := FALSE;
   AxisNuw.Axis[6].Pos8.Position := 0.0;
   AxisNuw.Axis[6].Pos8.Speed := 0;
   AxisNuw.Axis[6].Pos8.Reached := FALSE;
   AxisNuw.Axis[6].Pos9.Position := 0.0;
   AxisNuw.Axis[6].Pos9.Speed := 0;
   AxisNuw.Axis[6].Pos9.Reached := FALSE;
   AxisNuw.Axis[6].Pos10.Position := 0.0;
   AxisNuw.Axis[6].Pos10.Speed := 0;
   AxisNuw.Axis[6].Pos10.Reached := FALSE;
   AxisNuw.Axis[6].Pos11.Position := 0.0;
   AxisNuw.Axis[6].Pos11.Speed := 0;
   AxisNuw.Axis[6].Pos11.Reached := FALSE;
   AxisNuw.Axis[6].Pos12.Position := 0.0;
   AxisNuw.Axis[6].Pos12.Speed := 0;
   AxisNuw.Axis[6].Pos12.Reached := FALSE;
   AxisNuw.Axis[6].Pos13.Position := 0.0;
   AxisNuw.Axis[6].Pos13.Speed := 0;
   AxisNuw.Axis[6].Pos13.Reached := FALSE;
   AxisNuw.Axis[6].Pos14.Position := 0.0;
   AxisNuw.Axis[6].Pos14.Speed := 0;
   AxisNuw.Axis[6].Pos14.Reached := FALSE;
   AxisNuw.Axis[6].Pos15.Position := 0.0;
   AxisNuw.Axis[6].Pos15.Speed := 0;
   AxisNuw.Axis[6].Pos15.Reached := FALSE;
   AxisNuw.Axis[6].Pos16.Position := 0.0;
   AxisNuw.Axis[6].Pos16.Speed := 0;
   AxisNuw.Axis[6].Pos16.Reached := FALSE;
   AxisNuw.Axis[6].Pos17.Position := 0.0;
   AxisNuw.Axis[6].Pos17.Speed := 0;
   AxisNuw.Axis[6].Pos17.Reached := FALSE;
   AxisNuw.Axis[6].Pos18.Position := 0.0;
   AxisNuw.Axis[6].Pos18.Speed := 0;
   AxisNuw.Axis[6].Pos18.Reached := FALSE;
   AxisNuw.Axis[6].Pos19.Position := 0.0;
   AxisNuw.Axis[6].Pos19.Speed := 0;
   AxisNuw.Axis[6].Pos19.Reached := FALSE;
   AxisNuw.Axis[6].Pos20.Position := 0.0;
   AxisNuw.Axis[6].Pos20.Speed := 0;
   AxisNuw.Axis[6].Pos20.Reached := FALSE;
   AxisNuw.Axis[6].Pos21.Position := 0.0;
   AxisNuw.Axis[6].Pos21.Speed := 0;
   AxisNuw.Axis[6].Pos21.Reached := FALSE;
   AxisNuw.Axis[6].Pos22.Position := 0.0;
   AxisNuw.Axis[6].Pos22.Speed := 0;
   AxisNuw.Axis[6].Pos22.Reached := FALSE;
   AxisNuw.Axis[6].Pos23.Position := 0.0;
   AxisNuw.Axis[6].Pos23.Speed := 0;
   AxisNuw.Axis[6].Pos23.Reached := FALSE;
   AxisNuw.Axis[6].Pos24.Position := 0.0;
   AxisNuw.Axis[6].Pos24.Speed := 0;
   AxisNuw.Axis[6].Pos24.Reached := FALSE;
   AxisNuw.Axis[6].Pos25.Position := 0.0;
   AxisNuw.Axis[6].Pos25.Speed := 0;
   AxisNuw.Axis[6].Pos25.Reached := FALSE;
   AxisNuw.Axis[6].Pos26.Position := 0.0;
   AxisNuw.Axis[6].Pos26.Speed := 0;
   AxisNuw.Axis[6].Pos26.Reached := FALSE;
   AxisNuw.Axis[6].Pos27.Position := 0.0;
   AxisNuw.Axis[6].Pos27.Speed := 0;
   AxisNuw.Axis[6].Pos27.Reached := FALSE;
   AxisNuw.Axis[6].Pos28.Position := 0.0;
   AxisNuw.Axis[6].Pos28.Speed := 0;
   AxisNuw.Axis[6].Pos28.Reached := FALSE;
   AxisNuw.Axis[6].Pos29.Position := 0.0;
   AxisNuw.Axis[6].Pos29.Speed := 0;
   AxisNuw.Axis[6].Pos29.Reached := FALSE;
   AxisNuw.Axis[6].Pos30.Position := 0.0;
   AxisNuw.Axis[6].Pos30.Speed := 0;
   AxisNuw.Axis[6].Pos30.Reached := FALSE;
   AxisNuw.Axis[7].Pos1.Position := 0.0;
   AxisNuw.Axis[7].Pos1.Speed := 0;
   AxisNuw.Axis[7].Pos1.Reached := FALSE;
   AxisNuw.Axis[7].Pos2.Position := 0.0;
   AxisNuw.Axis[7].Pos2.Speed := 0;
   AxisNuw.Axis[7].Pos2.Reached := FALSE;
   AxisNuw.Axis[7].Pos3.Position := 0.0;
   AxisNuw.Axis[7].Pos3.Speed := 0;
   AxisNuw.Axis[7].Pos3.Reached := FALSE;
   AxisNuw.Axis[7].Pos4.Position := 0.0;
   AxisNuw.Axis[7].Pos4.Speed := 0;
   AxisNuw.Axis[7].Pos4.Reached := FALSE;
   AxisNuw.Axis[7].Pos5.Position := 0.0;
   AxisNuw.Axis[7].Pos5.Speed := 0;
   AxisNuw.Axis[7].Pos5.Reached := FALSE;
   AxisNuw.Axis[7].Pos6.Position := 0.0;
   AxisNuw.Axis[7].Pos6.Speed := 0;
   AxisNuw.Axis[7].Pos6.Reached := FALSE;
   AxisNuw.Axis[7].Pos7.Position := 0.0;
   AxisNuw.Axis[7].Pos7.Speed := 0;
   AxisNuw.Axis[7].Pos7.Reached := FALSE;
   AxisNuw.Axis[7].Pos8.Position := 0.0;
   AxisNuw.Axis[7].Pos8.Speed := 0;
   AxisNuw.Axis[7].Pos8.Reached := FALSE;
   AxisNuw.Axis[7].Pos9.Position := 0.0;
   AxisNuw.Axis[7].Pos9.Speed := 0;
   AxisNuw.Axis[7].Pos9.Reached := FALSE;
   AxisNuw.Axis[7].Pos10.Position := 0.0;
   AxisNuw.Axis[7].Pos10.Speed := 0;
   AxisNuw.Axis[7].Pos10.Reached := FALSE;
   AxisNuw.Axis[7].Pos11.Position := 0.0;
   AxisNuw.Axis[7].Pos11.Speed := 0;
   AxisNuw.Axis[7].Pos11.Reached := FALSE;
   AxisNuw.Axis[7].Pos12.Position := 0.0;
   AxisNuw.Axis[7].Pos12.Speed := 0;
   AxisNuw.Axis[7].Pos12.Reached := FALSE;
   AxisNuw.Axis[7].Pos13.Position := 0.0;
   AxisNuw.Axis[7].Pos13.Speed := 0;
   AxisNuw.Axis[7].Pos13.Reached := FALSE;
   AxisNuw.Axis[7].Pos14.Position := 0.0;
   AxisNuw.Axis[7].Pos14.Speed := 0;
   AxisNuw.Axis[7].Pos14.Reached := FALSE;
   AxisNuw.Axis[7].Pos15.Position := 0.0;
   AxisNuw.Axis[7].Pos15.Speed := 0;
   AxisNuw.Axis[7].Pos15.Reached := FALSE;
   AxisNuw.Axis[7].Pos16.Position := 0.0;
   AxisNuw.Axis[7].Pos16.Speed := 0;
   AxisNuw.Axis[7].Pos16.Reached := FALSE;
   AxisNuw.Axis[7].Pos17.Position := 0.0;
   AxisNuw.Axis[7].Pos17.Speed := 0;
   AxisNuw.Axis[7].Pos17.Reached := FALSE;
   AxisNuw.Axis[7].Pos18.Position := 0.0;
   AxisNuw.Axis[7].Pos18.Speed := 0;
   AxisNuw.Axis[7].Pos18.Reached := FALSE;
   AxisNuw.Axis[7].Pos19.Position := 0.0;
   AxisNuw.Axis[7].Pos19.Speed := 0;
   AxisNuw.Axis[7].Pos19.Reached := FALSE;
   AxisNuw.Axis[7].Pos20.Position := 0.0;
   AxisNuw.Axis[7].Pos20.Speed := 0;
   AxisNuw.Axis[7].Pos20.Reached := FALSE;
   AxisNuw.Axis[7].Pos21.Position := 0.0;
   AxisNuw.Axis[7].Pos21.Speed := 0;
   AxisNuw.Axis[7].Pos21.Reached := FALSE;
   AxisNuw.Axis[7].Pos22.Position := 0.0;
   AxisNuw.Axis[7].Pos22.Speed := 0;
   AxisNuw.Axis[7].Pos22.Reached := FALSE;
   AxisNuw.Axis[7].Pos23.Position := 0.0;
   AxisNuw.Axis[7].Pos23.Speed := 0;
   AxisNuw.Axis[7].Pos23.Reached := FALSE;
   AxisNuw.Axis[7].Pos24.Position := 0.0;
   AxisNuw.Axis[7].Pos24.Speed := 0;
   AxisNuw.Axis[7].Pos24.Reached := FALSE;
   AxisNuw.Axis[7].Pos25.Position := 0.0;
   AxisNuw.Axis[7].Pos25.Speed := 0;
   AxisNuw.Axis[7].Pos25.Reached := FALSE;
   AxisNuw.Axis[7].Pos26.Position := 0.0;
   AxisNuw.Axis[7].Pos26.Speed := 0;
   AxisNuw.Axis[7].Pos26.Reached := FALSE;
   AxisNuw.Axis[7].Pos27.Position := 0.0;
   AxisNuw.Axis[7].Pos27.Speed := 0;
   AxisNuw.Axis[7].Pos27.Reached := FALSE;
   AxisNuw.Axis[7].Pos28.Position := 0.0;
   AxisNuw.Axis[7].Pos28.Speed := 0;
   AxisNuw.Axis[7].Pos28.Reached := FALSE;
   AxisNuw.Axis[7].Pos29.Position := 0.0;
   AxisNuw.Axis[7].Pos29.Speed := 0;
   AxisNuw.Axis[7].Pos29.Reached := FALSE;
   AxisNuw.Axis[7].Pos30.Position := 0.0;
   AxisNuw.Axis[7].Pos30.Speed := 0;
   AxisNuw.Axis[7].Pos30.Reached := FALSE;
   AxisNuw.Axis[8].Pos1.Position := 0.0;
   AxisNuw.Axis[8].Pos1.Speed := 0;
   AxisNuw.Axis[8].Pos1.Reached := FALSE;
   AxisNuw.Axis[8].Pos2.Position := 0.0;
   AxisNuw.Axis[8].Pos2.Speed := 0;
   AxisNuw.Axis[8].Pos2.Reached := FALSE;
   AxisNuw.Axis[8].Pos3.Position := 0.0;
   AxisNuw.Axis[8].Pos3.Speed := 0;
   AxisNuw.Axis[8].Pos3.Reached := FALSE;
   AxisNuw.Axis[8].Pos4.Position := 0.0;
   AxisNuw.Axis[8].Pos4.Speed := 0;
   AxisNuw.Axis[8].Pos4.Reached := FALSE;
   AxisNuw.Axis[8].Pos5.Position := 0.0;
   AxisNuw.Axis[8].Pos5.Speed := 0;
   AxisNuw.Axis[8].Pos5.Reached := FALSE;
   AxisNuw.Axis[8].Pos6.Position := 0.0;
   AxisNuw.Axis[8].Pos6.Speed := 0;
   AxisNuw.Axis[8].Pos6.Reached := FALSE;
   AxisNuw.Axis[8].Pos7.Position := 0.0;
   AxisNuw.Axis[8].Pos7.Speed := 0;
   AxisNuw.Axis[8].Pos7.Reached := FALSE;
   AxisNuw.Axis[8].Pos8.Position := 0.0;
   AxisNuw.Axis[8].Pos8.Speed := 0;
   AxisNuw.Axis[8].Pos8.Reached := FALSE;
   AxisNuw.Axis[8].Pos9.Position := 0.0;
   AxisNuw.Axis[8].Pos9.Speed := 0;
   AxisNuw.Axis[8].Pos9.Reached := FALSE;
   AxisNuw.Axis[8].Pos10.Position := 0.0;
   AxisNuw.Axis[8].Pos10.Speed := 0;
   AxisNuw.Axis[8].Pos10.Reached := FALSE;
   AxisNuw.Axis[8].Pos11.Position := 0.0;
   AxisNuw.Axis[8].Pos11.Speed := 0;
   AxisNuw.Axis[8].Pos11.Reached := FALSE;
   AxisNuw.Axis[8].Pos12.Position := 0.0;
   AxisNuw.Axis[8].Pos12.Speed := 0;
   AxisNuw.Axis[8].Pos12.Reached := FALSE;
   AxisNuw.Axis[8].Pos13.Position := 0.0;
   AxisNuw.Axis[8].Pos13.Speed := 0;
   AxisNuw.Axis[8].Pos13.Reached := FALSE;
   AxisNuw.Axis[8].Pos14.Position := 0.0;
   AxisNuw.Axis[8].Pos14.Speed := 0;
   AxisNuw.Axis[8].Pos14.Reached := FALSE;
   AxisNuw.Axis[8].Pos15.Position := 0.0;
   AxisNuw.Axis[8].Pos15.Speed := 0;
   AxisNuw.Axis[8].Pos15.Reached := FALSE;
   AxisNuw.Axis[8].Pos16.Position := 0.0;
   AxisNuw.Axis[8].Pos16.Speed := 0;
   AxisNuw.Axis[8].Pos16.Reached := FALSE;
   AxisNuw.Axis[8].Pos17.Position := 0.0;
   AxisNuw.Axis[8].Pos17.Speed := 0;
   AxisNuw.Axis[8].Pos17.Reached := FALSE;
   AxisNuw.Axis[8].Pos18.Position := 0.0;
   AxisNuw.Axis[8].Pos18.Speed := 0;
   AxisNuw.Axis[8].Pos18.Reached := FALSE;
   AxisNuw.Axis[8].Pos19.Position := 0.0;
   AxisNuw.Axis[8].Pos19.Speed := 0;
   AxisNuw.Axis[8].Pos19.Reached := FALSE;
   AxisNuw.Axis[8].Pos20.Position := 0.0;
   AxisNuw.Axis[8].Pos20.Speed := 0;
   AxisNuw.Axis[8].Pos20.Reached := FALSE;
   AxisNuw.Axis[8].Pos21.Position := 0.0;
   AxisNuw.Axis[8].Pos21.Speed := 0;
   AxisNuw.Axis[8].Pos21.Reached := FALSE;
   AxisNuw.Axis[8].Pos22.Position := 0.0;
   AxisNuw.Axis[8].Pos22.Speed := 0;
   AxisNuw.Axis[8].Pos22.Reached := FALSE;
   AxisNuw.Axis[8].Pos23.Position := 0.0;
   AxisNuw.Axis[8].Pos23.Speed := 0;
   AxisNuw.Axis[8].Pos23.Reached := FALSE;
   AxisNuw.Axis[8].Pos24.Position := 0.0;
   AxisNuw.Axis[8].Pos24.Speed := 0;
   AxisNuw.Axis[8].Pos24.Reached := FALSE;
   AxisNuw.Axis[8].Pos25.Position := 0.0;
   AxisNuw.Axis[8].Pos25.Speed := 0;
